      120: SR50_Hori_servo_ctrl.Position:=(OP50_HORI_SERVO_PICK_POS+OP50_Hori_Ser_Jerk_Pos);
	  	   SR50_HORI_servo_ctrl.ABSmove_Start := TRUE;
		   OP50_AutoSeq:=130;

    		   
      130:  SR50_HORI_servo_ctrl.ABSmove_Start := 0;
			SR50_VERT_servo_ctrl.ABSmove_Start := TRUE;	   //MOVING VERTICL SERVO TO SAFE-WORK
            IF OP50_VERT_SERVO_ON_SFE_WRK  THEN
    	      SR50_VERT_servo_ctrl.ABSmove_Start := FALSE;
			  OP50_pick_done:=TRUE;
              OP50_AutoSeq:=140;   
    		END_IF
    		   
      140:  IF (NOT OP50_Gripper_LH_State AND OP50_Grip_LH_Bypass ) AND OP50_Gripper_RH_State THEN  
    			OP50_AutoSeq:=150;
			ELSIF (NOT OP50_Gripper_RH_State AND OP50_Grip_RH_Bypass) AND OP50_Gripper_LH_State THEN
				OP50_AutoSeq:=150;
			ELSIF OP50_Gripper_LH_State AND OP50_Gripper_RH_State THEN  
    			OP50_AutoSeq:=150;
			ELSIF (NOT OP50_Gripper_LH_State AND NOT OP50_Grip_LH_Bypass) OR (NOT OP50_Gripper_RH_State AND NOT OP50_Grip_RH_Bypass) THEN	
				OP50_AutoSeq:=220;
			ELSIF OP50_Grip_LH_Bypass AND OP50_Grip_RH_Bypass THEN
				OP50_AutoSeq:=250;
			END_IF	 
    	    		  
       150:  IF OP50_VERT_SERVO_ON_SFE_WRK  THEN // FEEDING PLACE POSITION TO HORIZONTAL SERVO
    		  SR50_Hori_servo_ctrl.Position:=OP50_HORI_SERVO_PLACE_POS;
              OP50_AutoSeq:=160;				 
    		 END_IF
    		   
       160:  SR50_HORI_servo_ctrl.ABSmove_Start := TRUE;    // MOVING HORIZONTAL SERVO TO PLACE POSITION
    		   IF OP50_HORI_SERVO_ON_WRK_PLACE THEN
    			 SR50_HORI_servo_ctrl.ABSmove_Start := FALSE;
    			 OP50_AutoSeq:=170;
    		   END_IF
       
       170: PAP_CYC_VAR:=0;
			IF OP50_HORI_SERVO_ON_WRK_PLACE AND NOT SR50_VERT_servo_ctrl.ABSmove_Start AND OP50_VERT_SERVO_ON_SFE_WRK AND OP50_STN_ENABLE THEN
    	   	  SR50_Vert_servo_ctrl.Position:=OP50_VERT_SERVO_PLACE_POS;
              OP50_AutoSeq:=175;		
      		END_IF
			
	   175: IF FIXTURE_LH<>40 AND FIXTURE_RH<>40 THEN
		   		OP50_AutoSeq:=250;	
			ELSIF FIXTURE_LH<>40 OR FIXTURE_RH<>40 THEN
				OP50_AutoSeq:=260;	
			ELSE
				OP50_AutoSeq:=180;		
	  	    END_IF
    		
       180: SR50_VERT_servo_ctrl.ABSmove_Start := TRUE; //MOVING VERTICAL SERVO TO PLACE POSITION
    		IF OP50_VERT_SERVO_ON_WRK_PLACE THEN
    			SR50_VERT_servo_ctrl.ABSmove_Start := FALSE;			
				OP50_AutoSeq:=190;				
    		END_IF	
			
       190: IF FIXTURE_LH=40 AND NOT OP50_Grip_LH_Bypass THEN 
				OP50_Gripper_LH_Close:=TRUE;	
			END_IF	
			IF FIXTURE_RH=40 AND NOT OP50_Grip_RH_Bypass THEN 
				OP50_Gripper_RH_Close:=TRUE;	
			END_IF		
			IF Gripper_Aft_Place_Delay.Q THEN	
				OP50_AutoSeq:=200;
			END_IF
			OP50_CURR_MOVER 			:= OP50_STN_MOVER;
			
       200:  //MOVING BACK TO VERTICAL SERVO SAFE POSITION
    		 IF OP50_VERT_SERVO_ON_WRK_PLACE AND NOT SR50_VERT_servo_ctrl.ABSmove_Start THEN
    		   SR50_Vert_servo_ctrl.Position:=OP50_VERT_SERVO_SFE_WRK_POS;
               OP50_AutoSeq:=201; 			   
    		 END_IF
 
	   201: IF Dry_Run THEN
				OP50_AutoSeq:=210; 
			END_IF
			IF  FIXTURE_LH=40 AND FIXTURE_RH=40 THEN
				MOVER_CMP_STATUS[OP50_CURR_MOVER][1]:=50 ;
				MOVER_CMP_STATUS[OP50_CURR_MOVER][2]:=50 ;
				OP50_AutoSeq:=210;
			ELSIF FIXTURE_LH=40 THEN
				MOVER_CMP_STATUS[OP50_CURR_MOVER][1]:=50 ;
				OP50_AutoSeq:=210;
			ELSIF FIXTURE_RH=40 THEN
				MOVER_CMP_STATUS[OP50_CURR_MOVER][2]:=50 ;
				OP50_AutoSeq:=210;
			END_IF		    		 
       210:	  //PROCEEDING FOR NEXT CYCLE
			   SR50_VERT_servo_ctrl.ABSmove_Start := TRUE;           
              IF OP50_VERT_SERVO_ON_SFE_WRK OR OP50_VERT_SERVO_ON_HOME THEN
    			  SR50_VERT_servo_ctrl.ABSmove_Start := FALSE;
				  OP50_STN_ENABLE:=0;				  	  
    			  IF OP50_Gripper_LH_State OR OP50_Gripper_RH_State THEN
    		  		OP50_AutoSeq:=220;
    			  ELSIF (MOVER_CMP_STATUS[OP50_STN_MOVER][1]=50 OR MOVER_CMP_STATUS[OP50_STN_MOVER][2]=50) OR Dry_Run THEN
					STATION_DONE[OP50_CURR_MOVER][OP50_XTS_POS_NO]			:= TRUE;
					IF MOVER_STP_NO[OP50_CURR_MOVER]<>((OP50_XTS_POS_NO*10)+1)THEN
						OP50_AutoSeq:=66;
					END_IF  
				  END_IF				  
    		  END_IF
    		  
       220:  IF (OP50_VERT_SERVO_ON_SFE_WRK OR OP50_VERT_SERVO_ON_HOME OR OP50_VERT_SERVO_ON_WRK_PICK OR OP50_VERT_SERVO_ON_WRK_PLACE) AND NOT SR50_HORI_servo_ctrl.ABSmove_Start AND (OP50_HORI_SERVO_ON_WRK_PLACE OR OP50_HORI_SERVO_ON_WRK_Pick OR OP50_HORI_SERVO_ON_HOME) THEN
    		  SR50_Hori_servo_ctrl.Position:=OP50_HORI_SERVO_SFE_WRK_POS;
			  SR50_Vert_servo_ctrl.Position:=OP50_VERT_SERVO_SFE_WRK_POS;	
              OP50_AutoSeq:=240;			  
    		 END_IF  
    	
       240: SR50_VERT_servo_ctrl.ABSmove_Start := TRUE;
	        IF OP50_VERT_SERVO_ON_SFE_WRK THEN
				SR50_HORI_servo_ctrl.ABSmove_Start := TRUE;
				OP50_AutoSeq:=242;
			 END_IF
			 
	  242: IF OP50_HORI_SERVO_ON_SFE_WRK THEN
    	  	 SR50_HORI_servo_ctrl.ABSmove_Start := FALSE;
      		 OP50_Gripper_RH_Close:=TRUE;	
    		 OP50_Gripper_LH_Close:=TRUE; 	
			 OP50_AutoSeq:=245;		   
      	   END_IF
	 
      245: IF OP50_HORI_SERVO_ON_SFE_WRK AND (NOT OP50_Gripper_LH_State AND NOT OP50_Gripper_RH_State) THEN
    		    OP50_Size_Rej_Complete:=1;
				OP50_AutoSeq:=66;
    	   END_IF
			 
	  250://MOVER_CMP_STATUS[OP50_CURR_MOVER][1]:=51;
		  //MOVER_CMP_STATUS[OP50_CURR_MOVER][2]:=51;
		  OP50_STN_ENABLE:=0;
		  IF (MOVER_CMP_STATUS[OP50_STN_MOVER][1]=51 AND MOVER_CMP_STATUS[OP50_STN_MOVER][2]=51) THEN
			MOVER_STP_NO[OP50_CURR_MOVER]	:= (OP160_XTS_POS_NO*10);
		  ELSE
			STATION_DONE[OP50_CURR_MOVER][OP50_XTS_POS_NO]			:= TRUE;
		  END_IF
		  IF MOVER_STP_NO[OP50_CURR_MOVER]<>((OP50_XTS_POS_NO*10)+1)THEN
			OP50_CURR_MOVER		:= 0;
		  OP50_AutoSeq:=170;	
 		END_IF
		
		
	   260: SR50_Hori_servo_ctrl.Position:=OP50_HORI_SERVO_SFE_WRK_POS;
			SR50_Hori_servo_ctrl.ABSmove_Start:=TRUE;
			IF OP50_HORI_SERVO_ON_SFE_WRK THEN
				OP50_AutoSeq:=270; 
			END_IF
			
	   270: IF FIXTURE_LH<>40 AND NOT OP50_Grip_LH_Bypass THEN
				OP50_Gripper_LH_Close:=TRUE;
				IF NOT OP50_Gripper_LH_State THEN
					OP50_AutoSeq:=280; 
				END_IF
			ELSE
				OP50_AutoSeq:=280;	
			END_IF	
			
	   280: IF FIXTURE_RH<>40 AND NOT OP50_Grip_RH_Bypass THEN
				OP50_Gripper_RH_Close:=TRUE;
				IF NOT OP50_Gripper_RH_State THEN
					OP50_AutoSeq:=290; 
				END_IF
			ELSE
				OP50_AutoSeq:=290;	
			END_IF	

	   290: SR50_Hori_servo_ctrl.Position:=OP50_HORI_SERVO_PLACE_POS;
			SR50_Hori_servo_ctrl.ABSmove_Start:=TRUE;
			IF OP50_HORI_SERVO_ON_WRK_PLACE THEN
				OP50_AutoSeq:=180;	
			END_IF
		
	 300: IF (OP50_HORI_SERVO_ON_SFE_WRK OR OP50_HORI_SERVO_ON_HOME OR OP50_HORI_SERVO_ON_SFE_WRK_PICK ) AND NOT SR50_HORI_servo_ctrl.ABSmove_Start AND OP50_Size_Rej THEN
		  		SR50_Hori_servo_ctrl.Position:=OP50_HORI_SERVO_PICK_POS;
				OP50_Size_Rej_Complete :=0;	
				OP50_Size_Rej          :=0;		
				OP50_AutoSeq:=310;
	       END_IF
		   
	  310: SR50_Hori_servo_ctrl.ABSmove_Start  := TRUE;
		   IF OP50_HORI_SERVO_ON_WRK_PICK THEN
		  		SR50_Vert_servo_ctrl.Position:=OP50_VERT_SERVO_PICK_POS;
				OP50_AutoSeq:=320;
	  	   END_IF
		   
	 320: SR50_VERT_servo_ctrl.ABSmove_Start := TRUE;
		  IF OP50_VERT_SERVO_ON_WRK_PICK THEN
		 	  OP50_Gripper_LH_Open:=OP50_LH_Size_NOK;
			  OP50_Gripper_RH_Open:=OP50_RH_Size_NOK;
			  IF Rejection_Grip_Delay.Q THEN
			  	OP50_AutoSeq:=220;
			  END_IF	
	 	  END_IF	
			
END_CASE

IF OP50_Size_Rej AND OP50_AutoRunning THEN
	OP50_AutoSeq:=300;
END_IF

OP50_STN_ENABLE:=OP50_Continous_Run;

Dry_Run:=All_Station_Dry_Run;
IF Dry_run THEN
	FIXTURE_LH :=40;	
    FIXTURE_RH :=40;
ELSE 
	FIXTURE_LH:=MOVER_CMP_STATUS[OP50_STN_MOVER][1];
	FIXTURE_RH:=MOVER_CMP_STATUS[OP50_STN_MOVER][2];
END_IF

Gripper_Delay(IN:=((OP50_Gripper_RH_State OR OP50_Grip_RH_Bypass) AND (OP50_Gripper_LH_State  OR OP50_Grip_LH_Bypass)),PT:=T#500MS);			
Gripper_pick_Delay(IN:=(OP50_AutoSeq=110),PT:=T#500MS);		
Gripper_Aft_pick_Delay (IN:=(OP50_AutoSeq=110),PT:=T#500MS); 
Gripper_Place_Delay	(IN:=(OP50_AutoSeq=110),PT:=T#500MS);	
Gripper_Aft_Place_Delay(IN:=(OP50_AutoSeq=190),PT:=T#700MS);
	
Rejection_Grip_Delay(IN:=OP50_Size_Rej_Complete,PT:=T#500MS);

del(IN:=tmp,PT:=T#700MS);
IF del.Q THEN
	tmp:=FALSE;
END_IF

//****************Cycle time block*********************************8

OP50_Cycle_Time_FB(i_b_startTime:=OP50_STN_ENABLE , i_b_stopTime:= NOT OP50_STN_ENABLE , o_t_StationTime=>OP50_Cycle_time );					
OP50_PAP_Cycle_Time_FB(i_b_startTime:=PAP_CYC_VAR , i_b_stopTime:= NOT PAP_CYC_VAR , o_t_StationTime=>OP50_PAP_Cycle_time );					
OP50_Overall_Cyc_Time:=OP50_Cycle_time+OP50_PAP_Cycle_time;


////################################ STATION ENABLE CONTION    ############################
OP50_STN_MOVER					:= MOVER_POSITION[OP50_XTS_POS_NO];
	
IF AUTO_WITH_XTS THEN
IF OP50_STN_MOVER>0 THEN
IF NOT(END_OF_CYCLE AND MOVER_CMP_STATUS[OP50_STN_MOVER][1]=5 AND MOVER_CMP_STATUS[OP50_STN_MOVER][2]=5)THEN	
	OP50_STN_ENABLE					:= MOVER_POS_RECHED[OP50_STN_MOVER] AND ((MOVER_CMP_STATUS[OP50_STN_MOVER][1]=40)OR 
										(MOVER_CMP_STATUS[OP50_STN_MOVER][2]=40))AND STATION_ENABLE_CONTROL;	
ELSE
	STATION_DONE[OP50_STN_MOVER][OP50_XTS_POS_NO]			:= TRUE;
END_IF
ELSE
	OP50_STN_ENABLE					:= FALSE;
END_IF	
END_IF

END_PROGRAM

// ---- POUs/Programs/OP50/OP50_Camera_FB.TcPOU
PROGRAM OP50_Camera_FB
VAR
	OP50_LH_Camera 			          : FB_Cognex_ProfiNET_1;

	OP50_LH_Acquisition_Status AT %I*    :Acquisition_Status;
	OP50_LH_Inspection_Status  AT %I*    :Inspection_Status;	
	OP50_LH_Acquisition_ID     AT %I*    :UINT;
	OP50_LH_Inspection_ID   	 AT %I*  :UINT;
	OP50_LH_Error_code      	 AT %I*  :UINT;
	OP50_LH_Current_Job_ID  	 AT %I*  :UINT;
	OP50_LH_Result_code     	 AT %I*  :UINT;
	OP50_LH_Cam_Result      	 AT %I*  :ARRAY[0..63] OF BYTE;	
	OP50_LH_Acquisition_Control AT %Q*  : Acquisition_Control;
	OP50_LH_Inspection_Control  AT %Q*  : Inspection_Control;
	OP50_LH_Command_word		AT %Q*  : UINT;
	OP50_LH_Union                       : UNION_64Byte;
	OP50_LH_Trigger_OK					: BOOL;
	
	OP50_RH_Camera 			          : FB_Cognex_ProfiNET_1;
	
	OP50_RH_Acquisition_Status AT %I*    :Acquisition_Status;
	OP50_RH_Inspection_Status  AT %I*    :Inspection_Status;	
	OP50_RH_Acquisition_ID     AT %I*    :UINT;
	OP50_RH_Inspection_ID   	 AT %I*  :UINT;
	OP50_RH_Error_code      	 AT %I*  :UINT;
	OP50_RH_Current_Job_ID  	 AT %I*  :UINT;
	OP50_RH_Result_code     	 AT %I*  :UINT;
	OP50_RH_Cam_Result      	 AT %I*  :ARRAY[0..63] OF BYTE;	
	OP50_RH_Acquisition_Control AT %Q*  : Acquisition_Control;
	OP50_RH_Inspection_Control  AT %Q*  : Inspection_Control;
	OP50_RH_Command_word		AT %Q*  : UINT;
	OP50_RH_Union                       : UNION_64Byte;
	OP50_RH_Trigger_OK					: BOOL;
END_VAR

OP50_LH_Camera (
	tTimeout:= , 
	sJob_Name:= , 
	camera_ready=> OP50_LH_Camera_Ready,
	Camera_online=> OP50_LH_Camera_Online,
	stCognex_record_status:=OP50_LH_Acquisition_Status, 
	Acquisition_ID:=OP50_LH_Acquisition_ID , 
	stCognex_Inspection_status:=OP50_LH_Inspection_Status, 
	Error_Code:=OP50_LH_Error_code , 
	wcommand_control_in:= OP50_LH_Current_Job_ID, 
	aResults_64_Bytes:= OP50_LH_Cam_Result, 
	number_of_inspections:=OP50_LH_Inspection_ID , 
	iresult_code:= OP50_LH_Result_code, 
	bTarget_job_ID:=OP50_LH_Target_Job_ID , 
	Error_Status_message=> OP50_LH_Error_status, 
	bError=> OP50_LH_Camera_Error, 
	stCognex_record_control=>OP50_LH_Acquisition_Control , 
	stCognex_inspection_control=>OP50_LH_Inspection_Control , 
	wCommandControl_out=>OP50_LH_Command_word , 
	aUser_data_64_Byte=> OP50_LH_Union.aArrayOfByte, 
	bJob_loading_completed=>OP50_LH_Job_Change_Complete , 
	bJob_load_failed=>OP50_LH_Job_Change_Error , 
	bInspection_Result_IO=>  OP50_LH_Trigger_OK, 
	bInspection_Result_NIO=> , 
	bTXTSM_Error_Job_Change=> OP50_LH_Job_Change_Error, 
	bPictureTakenComplete=> OP50_LH_Picture_Taken, 
	Loaded_Job_ID=>OP50_LH_Loaded_Job_ID	 , 
	bClear_Error:= HMI_Reset, 
	bJob_change_start:= OP50_LH_Camera_Job_Change_start, 
	TXTSM_camera_not_online=>OP50_LH_Camera_Error	 , 
	bTrigger_start:= OP50_LH_Camera_Trigger );
	
OP50_RH_Camera (
	tTimeout:= , 
	sJob_Name:= , 
	camera_ready=> OP50_RH_Camera_Ready,
	Camera_online=> OP50_RH_Camera_Online,
	stCognex_record_status:=OP50_RH_Acquisition_Status, 
	Acquisition_ID:=OP50_RH_Acquisition_ID , 
	stCognex_Inspection_status:=OP50_RH_Inspection_Status, 
	Error_Code:=OP50_RH_Error_code , 
	wcommand_control_in:= OP50_RH_Current_Job_ID, 
	aResults_64_Bytes:= OP50_RH_Cam_Result, 
	number_of_inspections:=OP50_RH_Inspection_ID , 
	iresult_code:= OP50_RH_Result_code, 
	bTarget_job_ID:=OP50_RH_Target_Job_ID , 
	Error_Status_message=> OP50_RH_Error_status, 
	bError=> OP50_RH_Camera_Error, 
	stCognex_record_control=>OP50_RH_Acquisition_Control , 
	stCognex_inspection_control=>OP50_RH_Inspection_Control , 
	wCommandControl_out=>OP50_RH_Command_word , 
	aUser_data_64_Byte=> OP50_RH_Union.aArrayOfByte, 
	bJob_loading_completed=>OP50_RH_Job_Change_Complete , 
	bJob_load_failed=>OP50_RH_Job_Change_Error , 
	bInspection_Result_IO=> OP50_RH_Trigger_OK , 
	bInspection_Result_NIO=> , 
	bTXTSM_Error_Job_Change=> OP50_RH_Job_Change_Error, 
	bPictureTakenComplete=> OP50_RH_Picture_Taken, 
	Loaded_Job_ID=>OP50_RH_Loaded_Job_ID	 , 
	bClear_Error:= HMI_Reset, 
	bJob_change_start:= OP50_RH_Camera_Job_Change_start, 
	TXTSM_camera_not_online=>OP50_RH_Camera_Error	 , 
	bTrigger_start:= OP50_RH_Camera_Trigger );

END_PROGRAM

// ---- POUs/Programs/OP50/OP50_Error.TcPOU
PROGRAM OP50_Error
VAR
	OP50_Step_Err_1: TON;
	OP50_Step_Err_2: TON;
	OP50_Step_Err_3: TON;
	OP50_Step_Err_4: TON;
	OP50_Step_Err_5: TON;
	OP50_Step_Err_6: TON;
	
	Gripper_ERR_Timer : TON;
END_VAR

// Set ERROR ACTIVE
IF ((OP50_GVL.OP50_ErrorWord_0<>0) OR (OP50_GVL.OP50_ErrorWord_1<>0) OR (OP50_GVL.OP50_ErrorWord_2<>0)) THEN
	OP50_GVL.OP50_ErrorActive:= TRUE;
END_IF

//Reset ErrorActive
IF OP50_HMI_Reset or HMI_Reset THEN 
	OP50_GVL.OP50_ErrorActive:= FALSE;
	OP50_GVL.OP50_ErrorWord_0:= 0;
	OP50_GVL.OP50_ErrorWord_1:= 0;
	OP50_GVL.OP50_ErrorWord_2:= 0;	
END_IF

// Auto Seq Step Error

//Horizontal Servo is not in home or safe-work position 
OP50_Step_Err_1(IN:=(OP50_GVL.OP50_AutoSeq=70) , PT:=T#5S , Q=> , ET=> );
IF (OP50_GVL.OP50_AutoSeq=70 AND OP50_Step_Err_1.Q) THEN
	OP50_GVL.OP50_ErrorWord_0.0:=TRUE;
END_IF


//Horizontal Servo not reaching pick position 
OP50_Step_Err_1(IN:=(OP50_GVL.OP50_AutoSeq=80) , PT:=T#5S , Q=> , ET=> );
IF (OP50_GVL.OP50_AutoSeq=80 AND NOT OP50_HORI_SERVO_ON_WRK_PICK AND OP50_Step_Err_1.Q) THEN
	OP50_GVL.OP50_ErrorWord_0.1:=TRUE;
END_IF

// Gripper is not closing
OP50_Step_Err_2(IN:=OP50_GVL.OP50_AutoSeq=82 , PT:=T#5S , Q=> , ET=> );
IF (OP50_GVL.OP50_AutoSeq=82 AND OP50_Step_Err_2.Q) THEN
	OP50_GVL.OP50_ErrorWord_0.2:=TRUE;
END_IF

// Vertical Servo not reaching work position 
OP50_Step_Err_3(IN:=OP50_GVL.OP50_AutoSeq=100 , PT:=T#5S , Q=> , ET=> );
IF (OP50_GVL.OP50_AutoSeq=100 AND OP50_Step_Err_3.Q) THEN
	OP50_GVL.OP50_ErrorWord_0.3:=TRUE;
END_IF

// Vertical Servo not reaching safe-work position 
OP50_Step_Err_3(IN:=OP50_GVL.OP50_AutoSeq=150 , PT:=T#5S , Q=> , ET=> );
IF (OP50_GVL.OP50_AutoSeq=150 AND OP50_Step_Err_3.Q) THEN
	OP50_GVL.OP50_ErrorWord_0.4:=TRUE;
END_IF

// Checking the gripper condition is opened or not
OP50_Step_Err_3(IN:=OP50_GVL.OP50_AutoSeq=140 , PT:=T#5S , Q=> , ET=> );
IF (OP50_GVL.OP50_AutoSeq=140 AND OP50_Step_Err_3.Q) THEN
	OP50_GVL.OP50_ErrorWord_0.5:=TRUE;
END_IF

//  Horizontal sevo not moving to place position
OP50_Step_Err_3(IN:=OP50_GVL.OP50_AutoSeq=160 , PT:=T#5S , Q=> , ET=> );
IF (OP50_GVL.OP50_AutoSeq=160 AND OP50_Step_Err_3.Q) THEN
	OP50_GVL.OP50_ErrorWord_0.6:=TRUE;
END_IF

//  Vertical sevo not moving to place position
OP50_Step_Err_3(IN:=OP50_GVL.OP50_AutoSeq=180 , PT:=T#5S , Q=> , ET=> );
IF (OP50_GVL.OP50_AutoSeq=180 AND OP50_Step_Err_3.Q) THEN
	OP50_GVL.OP50_ErrorWord_0.7:=TRUE;
END_IF

// Vertical Servo not reaching safe-work position 
OP50_Step_Err_3(IN:=OP50_GVL.OP50_AutoSeq=210 , PT:=T#5S , Q=> , ET=> );
IF (OP50_GVL.OP50_AutoSeq=210 AND OP50_Step_Err_3.Q) THEN
	OP50_GVL.OP50_ErrorWord_0.8:=TRUE;
END_IF

//  Horizontal sevo not moving to safe work position
OP50_Step_Err_3(IN:=OP50_GVL.OP50_AutoSeq=240 , PT:=T#5S , Q=> , ET=> );
IF (OP50_GVL.OP50_AutoSeq=240 AND OP50_Step_Err_3.Q) THEN
	OP50_GVL.OP50_ErrorWord_0.9:=TRUE;
END_IF

IF Gripper_ERR_Timer.Q THEN
	OP50_GVL.OP50_ErrorWord_0.10:=TRUE;
END_IF

Gripper_ERR_Timer(IN:=I50_LH_GRIP_CLSE_I1101_7 OR I50_RH_GRIP_CLSE_I1110_1,PT:=T#500MS);

END_PROGRAM

// ---- POUs/Programs/OP50/OP50_Initialize_Seq.TcPOU
PROGRAM OP50_Initialize_Seq
VAR
END_VAR

IF OP50_GIUDE_GRP_ctrl.Axis_In_Home AND OP50_GIUDE_GRP_ctrl.Axis_Home_Done AND (SR50_Vert_servo_ctrl.Axis_In_Home) AND OP50_HORI_SERVO_ON_HOME AND NOT I50_LH_GRIP_CLSE_I1101_7 AND  NOT I50_RH_GRIP_CLSE_I1110_1 THEN
	OP50_Temp_hmeOK:=TRUE;
	OP50_HomeRunning:=FALSE;
	OP50_Homing_Seq:=0;
ELSE
	OP50_Temp_hmeOK:=FALSE;	
END_IF

CASE OP50_Homing_Seq OF
	0: IF (OP50_AutoSelected AND NOT OP50_HomeRunning AND NOT OP50_ErrorActive AND NOT OP50_AutoRunning AND NOT OP50_StepRunning AND NOT OP50_Temp_hmeOK) THEN
		OP50_HomeRunning:=TRUE;
		OP50_Homing_Seq:=10;	
	   END_IF
	   
	10:IF (OP50_HomeRunning AND (OP50_HMI_Homing OR HMI_Reset ))THEN 
		IF (SR50_Vert_servo_ctrl.Axis_In_Home) THEN 
			SR50_Vert_servo_ctrl.Axis_Home_Cmd:=FALSE;
		    OP50_Homing_Seq:=20;
		ELSE
			SR50_Vert_servo_ctrl.Position:=0;
			SR50_Vert_servo_ctrl.Velocity:=100;
			SR50_Vert_servo_ctrl.ABSmove_Start:=TRUE;
			SR50_Vert_servo_ctrl.Axis_Home_Cmd:=TRUE;		
	    END_IF
	   END_IF	
	   
   20:  IF (OP50_HORI_SERVO_ON_HOME) THEN 
			SR50_Hori_servo_ctrl.Axis_Home_Cmd:=FALSE;
			OP50_Homing_Seq:=40;
		ELSE
			SR50_Hori_servo_ctrl.Position:=OP50_HORI_SERVO_HME_POS;
			SR50_Hori_servo_ctrl.Velocity:=100;
			SR50_Hori_servo_ctrl.ABSmove_Start:=TRUE;
	    END_IF
		
   40:  CR50_LH_Grip_Cyl.HomingCmd1:=1;
   		CR50_RH_Grip_Cyl.HomingCmd1:=1;
		IF CR50_LH_Grip_Cyl.HomingCmd1 AND CR50_RH_Grip_Cyl.HomingCmd1 THEN
   			OP50_Homing_Seq:=50;
		END_IF	
   
   45:	IF NOT I50_LH_GRIP_CLSE_I1101_7 AND OP50_Gripper_LH_Close THEN 
			OP50_Gripper_LH_State := FALSE;
			OP50_Homing_Seq:=50;
			OP50_Gripper_LH_Close := FALSE;
	    END_IF
				
   50: 	 OP50_Gripper_LH_State := FALSE;
   		 OP50_Gripper_RH_State := FALSE;
   		 OP50_Homing_Seq:=60;
	
   55: 	IF NOT I50_RH_GRIP_CLSE_I1110_1 AND OP50_Gripper_RH_Close THEN 
			OP50_Gripper_RH_State := FALSE;
			OP50_Homing_Seq:=60;
			OP50_Gripper_RH_Close := FALSE;
	    END_IF
		
   60: 	CR50_LH_Rej_Cyl.HomingCmd1:=TRUE;	
		IF CR50_LH_Rej_Cyl.Position1 THEN
			CR50_LH_Rej_Cyl.HomingCmd1:=FALSE;
			OP50_Homing_Seq:=70;
		END_IF
		
   70:	CR50_RH_Rej_Cyl.HomingCmd1:=TRUE;	
		IF CR50_RH_Rej_Cyl.Position1 THEN
			CR50_RH_Rej_Cyl.HomingCmd1:=FALSE;
			OP50_Homing_Seq:=75;
		END_IF
	
  75:	IF OP50_GIUDE_GRP_ctrl.Axis_In_Home AND OP50_GIUDE_GRP_ctrl.Axis_Home_Done THEN
	  		OP50_GIUDE_GRP_ctrl.Bsethome:=0;
			OP50_Homing_Seq:=80;
		ELSE
			OP50_GIUDE_GRP_ctrl.Bsethome:=1;
  		END_IF
	
   80:	OP50_Homing_Seq:=0;
		OP50_HomeRunning:=FALSE;
		OP50_HMI_Homing:=FALSE;
END_CASE

IF NOT OP50_HomeRunning THEN
	   	CR50_LH_Grip_Cyl.HomingCmd1:=0;
		CR50_LH_Rej_Cyl.HomingCmd1:=FALSE;
		CR50_RH_Rej_Cyl.HomingCmd1:=FALSE;
   		CR50_RH_Grip_Cyl.HomingCmd1:=0;
END_IF

END_PROGRAM

// ---- POUs/Programs/OP50/OP50_Conveyor_Cam_Seq.TcPOU
PROGRAM OP50_Conveyor_Cam_Seq
VAR
	OP50_Conveyor_FB	: Servo_Conveyor_FB;
	OP50_Camera_Trigger : BOOL;
	Conveyor_Track_Delay: TON;
	Conveyor_Track_OFF_Delay: TON;
	Conveyor_Continuous_Run: BOOL;
	Conveyor_Velocity_mode: BOOL;
	 OP50_Camera_Trigger_Ack : BOOL;
	Conv_Cam_Step: INT;
	OP50_Miss_Trigger	: BOOL;
	Conv_Temp: BOOL;
	Conv_Step_no: INT;
	Temp_Counter_LH: UINT;
	Temp_Counter_RH: UINT;
	Toggle_Pos_LH : R_TRIG;
	Toggle_Neg_LH : F_TRIG;
	Toggle_Pos_RH : R_TRIG;
	Toggle_Neg_RH : F_TRIG;
	LH_Cam_Completed : BOOL;
	RH_Cam_Completed : BOOL;
	Drum_Jam_Timer	 : TON;
	Toggle_Neg: INT;
	OP50_Camera_Bypass : BOOL;
		Control : BOOL;
END_VAR

Toggle_Pos_LH(CLK:=OP50_Camera_FB.OP50_LH_Inspection_Status.Inspection_Completed);
Toggle_Neg_LH(CLK:=OP50_Camera_FB.OP50_LH_Inspection_Status.Inspection_Completed);
Toggle_Pos_RH(CLK:=OP50_Camera_FB.OP50_RH_Inspection_Status.Inspection_Completed);
Toggle_Neg_RH(CLK:=OP50_Camera_FB.OP50_RH_Inspection_Status.Inspection_Completed);

IF Toggle_Pos_LH.Q OR Toggle_Neg_LH.Q THEN
	LH_Cam_Completed:=1;	
END_IF
IF Toggle_Pos_RH.Q OR Toggle_Neg_RH.Q THEN
	RH_Cam_Completed:=1;	
END_IF


IF MANUAL_SELECTED AND OP50_ManualSelected THEN               
	IF I50_DRUM_CONV_REV_I306_3 THEN
		SR50_Conv_servo_status.targetVelocity:=OP50_Conv_Rev_Speed_6_3;
		SR50_Conv_servo_status.moveVelocity:=I50_DRUM_CONV_REV_I306_3;
 	ELSIF I50_DRUM_CONV_FWD_I306_4 THEN
		SR50_Conv_servo_status.targetVelocity:=OP50_Conv_Fwd_Speed_7_89;
		SR50_Conv_servo_status.moveVelocity:=I50_DRUM_CONV_FWD_I306_4;	
	ELSE 	
		SR50_Conv_servo_status.moveVelocity:=0;   	
	END_IF  	
END_IF

IF OP50_Model='6.3' THEN
	OP50_Conv_Fwd_Time:=OP50_Conv_Fwd_Time_6_3;
	OP50_Conv_Rev_Time:=OP50_Conv_Rev_Time_6_3;
	OP50_Conveyor_FWD_Speed:= OP50_Conv_Fwd_Speed_6_3;
	OP50_Conveyor_REV_Speed:= OP50_Conv_Rev_Speed_6_3;
END_IF

IF OP50_Model='7.89' THEN
	OP50_Conv_Fwd_Time:=OP50_Conv_Fwd_Time_7_89;
	OP50_Conv_Rev_Time:=OP50_Conv_Rev_Time_7_89;
	OP50_Conveyor_FWD_Speed:= OP50_Conv_Fwd_Speed_7_89;
	OP50_Conveyor_REV_Speed:= OP50_Conv_Rev_Speed_7_89;
END_IF

Conveyor_Velocity_mode:=1;

OP50_Conveyor_FB(
	Conveyor_Prgrm_Start:= OP50_AutoRunning, 
	Conveyor_Prgrm_Reset:= , 
	Conveyor_Continuous_Run:= Conveyor_Continuous_Run, 
	Camera_Trigger_OK := OP50_Camera_Done OR OP50_Camera_Bypass, 
	Fwd_Time_IP:= OP50_Conv_Fwd_Time, 
	Rev_Time_IP:= OP50_Conv_Rev_Time, 
	Track_Overflow := Conveyor_Track_OFF_Delay.Q, 
	Track_Sensor_FB := Conveyor_Track_Delay.Q,
	Conveyor_FWD_Position	:= OP50_Conv_Fwd_Pos,
    Conveyor_REV_Position	:= OP50_Conv_Rev_Pos,
    Velocity_mode			:= Conveyor_Velocity_mode,	
	Conveyor_FWD_Speed:=OP50_Conveyor_FWD_Speed , 
	Conveyor_REV_Speed:=OP50_Conveyor_REV_Speed , 
	LH_Work_Sensor:=CR50_LH_Rej_Cyl.Sensor2 , 
	LH_Home_Sensor:=CR50_LH_Rej_Cyl.Sensor1 , 
	RH_Work_Sensor:=CR50_RH_Rej_Cyl.Sensor2 , 
	RH_Home_Sensor:=CR50_RH_Rej_Cyl.Sensor1 , 
	LH_Camera_OK:=  OP50_LH_Camera_OK OR OP50_Camera_Bypass, 
	LH_Camera_NOK:= OP50_LH_Camera_NOK, 
	RH_Camera_OK:=  OP50_RH_Camera_OK OR OP50_Camera_Bypass, 
	RH_Camera_NOK:= OP50_RH_Camera_NOK,
	Step_Num => Conv_Step_no,
	Camera_Trigger_Ack=> OP50_Camera_Trigger_Ack, 
	Camera_trigger:= OP50_Camera_Trigger,
	Drum_ON=> O50_DRUM_MTR_FWD_Q305_5, 
	LH_Work_Coil=>CR50_LH_Rej_Cyl.AutoCmd2 , 
	LH_Home_Coil=>CR50_LH_Rej_Cyl.AutoCmd1 , 
	RH_Work_Coil=>CR50_RH_Rej_Cyl.AutoCmd2,
	RH_Home_Coil=>CR50_RH_Rej_Cyl.AutoCmd1,
	Ready_to_Pick=> OP50_pick_ready , 
	Pick_Done:=     OP50_pick_done , 
	One_Cycle		:= OP50_One_Cycle,
	Conveyor_Servo_Control_Structure:= SR50_CONV_servo_ctrl );

Conveyor_Track_Delay(IN:= NOT I50_DRUM_FEED_CONV1_OVERFLW_I1101_0 OR NOT I50_DRUM_FEED_CONV2_OVERFLW_I1101_1,PT:=INT_TO_TIME(OP50_Drum_ON_Time));	
Conveyor_Track_OFF_Delay(IN:=I50_DRUM_FEED_CONV1_OVERFLW_I1101_0 AND I50_DRUM_FEED_CONV2_OVERFLW_I1101_1,PT:=INT_TO_TIME(OP50_Drum_OFF_Time));  
	
IF 	OP50_AutoRunning OR Conv_Temp THEN
	IF Conveyor_Track_OFF_Delay.Q THEN
		O50_DRUM_MTR_FWD_Q305_5:=0;
	END_IF
	//IF Conveyor_Track_Delay.Q THEN
	//	O50_DRUM_MTR_FWD_Q305_5:=1;
	//END_IF
	O50_AIR_PURGE_ON_Q1153_4:=1;
	O50_DRUM_RUN_IND_Q306_2:=O50_DRUM_MTR_FWD_Q305_5;
ELSE
	O50_DRUM_RUN_IND_Q306_2:=I50_DRUM_OFF_ON_I306_2;
	O50_DRUM_MTR_FWD_Q305_5:=I50_DRUM_OFF_ON_I306_2;
	O50_AIR_PURGE_ON_Q1153_4:=I50_DRUM_OFF_ON_I306_2;
END_IF

IF (NOT OP50_AutoRunning OR (NOT OP50_LH_Camera_Online OR NOT OP50_RH_Camera_Online)) AND NOT OP50_Camera_Bypass THEN
	Conv_Cam_Step:=10;
END_IF 

CASE Conv_Cam_Step OF
	10: 	OP50_LH_Camera_OK :=0;
            OP50_LH_Camera_NOK:=0;
	        OP50_RH_Camera_OK :=0;
	        OP50_RH_Camera_NOK:=0;
			LH_Cam_Completed  :=0;
			RH_Cam_Completed  :=0;			
			OP50_Camera_Done	:=0;
			OP50_LH_Clr_OK 		:=0;
		    OP50_RH_Clr_OK 		:=0;		
			OP50_LH_Size_OK		:=0;
		    OP50_RH_Size_OK		:=0;	
			Conv_Cam_Step		:=11;	
	
	11: IF ((OP50_Camera_Trigger AND (NOT OP50_Camera_Done)) OR OP50_Miss_Trigger) AND NOT OP50_Camera_Bypass THEN
			OP50_LH_Camera_Trigger:=1;
			OP50_RH_Camera_Trigger:=1;
			Conv_Cam_Step		  :=15;	
		END_IF

	15:	IF LH_Cam_Completed AND RH_Cam_Completed THEN// (NOT OP50_LH_Camera_Trigger) AND (NOT OP50_RH_Camera_Trigger) THEN //(Temp_Counter_LH<OP50_Camera_FB.OP50_LH_Acquisition_ID AND Temp_Counter_RH<OP50_Camera_FB.OP50_RH_Acquisition_ID )THEN
			OP50_LH_Camera_Trigger:=0;
			OP50_RH_Camera_Trigger:=0;
			OP50_Camera_Trigger :=0;
			OP50_Miss_Trigger	:=0;
			Conv_Cam_Step:=25;
		END_IF  
	   
	25: IF OP50_Camera_FB.OP50_LH_Cam_Result[0]=1 AND OP50_Camera_FB.OP50_RH_Cam_Result[0]=1 THEN
			OP50_LH_Camera_OK:=1;
			OP50_RH_Camera_OK:=1;
			Conv_Cam_Step    :=50;
		ELSIF (OP50_Camera_FB.OP50_LH_Cam_Result[2]<>1 OR OP50_Camera_FB.OP50_RH_Cam_Result[2]<>1) THEN	
			OP50_One_Cycle  :=1;
			Conv_Cam_Step   :=50;
		ELSIF (OP50_Camera_FB.OP50_LH_Cam_Result[1]=1 OR OP50_Camera_FB.OP50_RH_Cam_Result[1]=1) AND (OP50_Camera_FB.OP50_LH_Cam_Result[2]=1 AND OP50_Camera_FB.OP50_RH_Cam_Result[2]=1) THEN					
			IF OP50_Camera_FB.OP50_LH_Cam_Result[0]=1 THEN
				OP50_LH_Camera_OK:=1;
			END_IF
			IF OP50_Camera_FB.OP50_RH_Cam_Result[0]=1 THEN
				OP50_RH_Camera_OK:=1;
			END_IF
			Conv_Cam_Step:=30;
		END_IF	
			
   30: 	IF OP50_Camera_FB.OP50_LH_Cam_Result[1]=1 THEN
	   		OP50_LH_Camera_NOK:=1;
  	    END_IF
		IF OP50_Camera_FB.OP50_RH_Cam_Result[1]=1 THEN
	   		OP50_RH_Camera_NOK:=1;
  	    END_IF
		Conv_Cam_Step:=50;
		
   50:  OP50_Camera_Done:=1;
   		Temp_Counter_LH:=OP50_Camera_FB.OP50_LH_Acquisition_ID;
		Temp_Counter_RH:=OP50_Camera_FB.OP50_RH_Acquisition_ID;
		IF Conv_Step_no>75 THEN
			Conv_Cam_Step   :=10;
			OP50_Camera_Done:=0;
		END_IF   
END_CASE


IF OP50_AutoRunning AND Control THEN
	Drum_Jam_Timer(IN:=(NOT I50_DRUM_FEED_CONV1_OVERFLW_I1101_0)OR(NOT I50_DRUM_FEED_CONV2_OVERFLW_I1101_1)); 
	Drum_Jam_Timer(PT:=T#40S);
	IF Drum_Jam_Timer.Q THEN
		OP50_ErrorActive:=1;
	END_IF
END_IF

END_PROGRAM

// ---- POUs/Programs/OP60/OP60_MAIN.TcPOU
PROGRAM OP60_MAIN
VAR
	OP60_Modeselection_FB: Mode_Selection_Block1;	
//	OP60_Cycle_Time: Cycle_Time_FB;
	//TP_100ms: TP;
	reset: BOOL;
	Gen_Timer: TON;
END_VAR

// Function Calling

OP60_Manual();
OP60_AUTOSEQUENCE();
OP60_Error();
OP60_Initialization_Seq();
op60_toolchangeover ();
//MOdeselection From HMI

IF (OP60_HMI_AutoMode AND NOT OP60_HMI_ManualMOde AND NOT OP60_HMI_StepMode) THEN
		OP60_Modeselection_FB.ModeWord:=1;
	ELSIF (NOT OP60_HMI_AutoMode AND OP60_HMI_ManualMOde AND NOT OP60_HMI_StepMode) THEN
		OP60_Modeselection_FB.ModeWord:=2;
	ELSIF  (NOT OP60_HMI_AutoMode AND NOT OP60_HMI_ManualMOde AND  OP60_HMI_StepMode) THEN
		OP60_Modeselection_FB.ModeWord:=3;
    ELSE   
		OP60_Modeselection_FB.ModeWord:=0;
END_IF

OP60_Safety_OK:=OperationEnable;

OP60_Modeselection_FB(
	ModeWord:= , 
	HomeConditionOK:=OP60_HomeConditionOK , 
	OperationEnable:=OP60_AutoSelected, 
	StartPB:=OP60_HMI_CycleStart , 
	SafetyAndNOError:= OP60_Safety_OK, 
	ModeAck:=TRUE , 
	HomingINProgress:=OP60_HomeRunning , 
	TempHomeOK:=OP60_Temp_hmeOK , 
	ResetPB:= , 
	AutoSelected=> OP60_AutoSelected, 
	ManualSelected=> OP60_ManualSelected, 
	StepSelected=>OP60_StepSelected , 
	ModeSelAck_Indication=> , 
	StatusDisplay=> , 
	AutoRunning:=OP60_AutoRunning, 
	StepRunning:=OP60_StepRunning , 
	StartEnable:=OP60_StartEnable  , 
	MachineStop:=OP60_Machine_Stop );

OP60_Safety_OK:=OperationEnable;	
	
IF OP60_AutoSelected OR OP60_ManualSelected AND NOT ( OP60_ErrorActive OR OP60_Safety_OK) THEN
	SR60_Vert_servo.bEnable:=TRUE;
ELSE
	SR60_Vert_servo.bEnable:=FALSE;
END_IF

IF OP60_GVL.SR60_Vert_servo.bAxisError OR NOT OP60_Safety_OK  THEN
	OP60_ErrorActive:=TRUE;
END_IF

IF OP60_Stop_Request AND NOT OP60_STN_ENABLE THEN
	OP60_Machine_Stop:=1;
END_IF
Gen_Timer(IN:=OP60_Machine_Stop,PT:=T#5S);
IF Gen_Timer.Q THEN
	OP60_Machine_Stop:=0;
END_IF

END_PROGRAM

// ---- POUs/Programs/OP60/OP60_MANUAL.TcPOU
PROGRAM OP60_MANUAL
VAR
	
    temp_safe:BOOL;
	enable:BOOL;
	reset:bool;
END_VAR


// IF MANUAL IS SELECTED 

//SR60_Vert_servo_ctrl.ABSmove_Start:=OP60_VERT_SERVO_STRT;
OP60_SERVO_POS_DONE:= SR60_Vert_servo_ctrl.pos_done;

IF In_Range(SR60_Vert_servo_status.actualPosition,OP60_VERT_SERVO_SFE_WRK_POS,3) THEN
	OP60_SERVO_ON_SFE_WRK := TRUE;
ELSE
	OP60_SERVO_ON_SFE_WRK := FALSE;
END_IF

IF In_Range(SR60_Vert_servo_status.actualPosition,OP60_VERT_SERVO_HME_POS,1) THEN
	OP60_SERVO_ON_HOME := TRUE;
ELSE
	OP60_SERVO_ON_HOME := FALSE;
END_IF

IF In_Range(SR60_Vert_servo_status.actualPosition,OP60_VERT_SERVO_WRK_POS_1,2) THEN
	OP60_SERVO_ON_WRK_1 := TRUE;
ELSE
	OP60_SERVO_ON_WRK_1 := FALSE;
END_IF

IF In_Range(SR60_Vert_servo_status.actualPosition,OP60_VERT_SERVO_WRK_POS_2,2) THEN
	OP60_SERVO_ON_WRK_2 := TRUE;
ELSE
	OP60_SERVO_ON_WRK_2 := FALSE;
END_IF

OP60_VERT_SERVO_SFE_WRK_POS   :=  OP60_HMI_Safe_Work;
OP60_VERT_SERVO_HME_POS       :=  OP60_HMI_Safe_Home;
OP60_VERT_SERVO_WRK_POS_2     :=  OP60_VERT_SERVO_WORK_POS;
OP60_VERT_SERVO_WRK_POS_1	  := (OP60_VERT_SERVO_WRK_POS_2-OP60_HMI_Servo_Pos_Offset);

SR60_Vert_servo(
	bAxis1_Ref_Switch:= , 
	bInit:= , 
	bErrorReset:= OP60_GVL.OP60_HMI_Reset OR Servo_Reset , 
	bEnable:=Servo_Enable, 
	bMoveVelocity:= , 
	bHalt:= , 
	bManualMode:= MANUAL_SELECTED AND OP60_ManualSelected, 
	fHomePos:= , 
	fOverride:= , 
	fTargetPosition:= SR60_Vert_servo_ctrl.Position, 
	fTargetVelocity:= SR60_Vert_servo_ctrl.Velocity, 
	fAcc:= , 
	fDec:= , 
	Servo_High_Limit:= OP60_HMI_High_Limit,	
	Servo_Low_Limit:=  OP60_HMI_Low_Limit,	
	Safe_move_Conditions:=Servo_Safety,
	Axis:=SR60_Vert_servo_Axis  , 
	bmove_home:=SR60_Vert_servo_ctrl.Axis_Home_Cmd ,
	baxis_in_home_pos=>SR60_Vert_servo_ctrl.Axis_In_Home ,
	HME_WRITE_ADD:= 16#5018, 
	bHome:=SR60_Vert_servo_ctrl.Bsethome , 
	bSetPosition:=SR60_Vert_servo_ctrl.BsetPos , 
	bMoveAbsolute:=SR60_Vert_servo_ctrl.ABSmove_Start , 
	bMoveTorque :=SR60_Vert_servo_ctrl.Torque_mode_Start,	
	bMoveRelative:=SR60_Vert_servo_ctrl.RELmove_Start , 
	stManualModeAxis:=SR60_Vert_servo_status , 
	sAxisState=>SR60_Vert_servo_ctrl.Axis_State , 
	bAxis_ready=>SR60_Vert_servo_ctrl.Axis_ready , 
	bAxisInPosition=> SR60_Vert_servo_ctrl.Axis_In_Pos, 
	bAxisError=>SR60_Vert_servo_ctrl.Axis_Error , 
	bAxisEnabled=> SR60_Vert_servo_ctrl.Axis_Enabled, 
	bAxisHomed=> SR60_Vert_servo_ctrl.Axis_reference, 
	bSetPositionDone=>   ,
    bsafe_to_move=>SR60_Vert_servo_ctrl.Safe_To_Move,  
	bABS_Pos_done=> SR60_Vert_servo_ctrl.pos_done,
	bHaltDone=> , 
	bSTOPDone=> , 
	bHomeDone=> , 
	bDone=> ,
	Actual_position=>SR60_Vert_servo_ctrl.Actual_Position ,  
	Actual_velocity=>SR60_Vert_servo_ctrl.Actual_Velocity , 
	Actual_Torque=> SR60_Vert_servo_ctrl.Actual_Torque);
	
IF MANUAL_SELECTED and OP60_ManualSelected THEN
	SR60_Vert_servo_status.targetVelocity:=250;	
END_IF	
	

OP60_LH_LVDT_VALUE := DINT_TO_REAL(OP60_LH)/10000;
OP60_RH_LVDT_VALUE := DINT_TO_REAL(OP60_RH)/10000;

END_PROGRAM

// ---- POUs/Programs/OP60/OP60_AUTOSEQUENCE.TcPOU
PROGRAM OP60_AUTOSEQUENCE
VAR

//INT

	OP60_FIXTURE_2					: INT;
	OP60_FIXTURE_1					: INT;	
	
// TIMER
	OP60_AFT_WRK_POS : TON;
	dry_run : BOOL;
	check: BOOL;

	OP60_STN_MOVER: INT;
	MOVER_POS_RECHED_R: R_TRIG;
	OP60_Cycle_Time_FB : FB_Cycletime;
END_VAR

VAR PERSISTENT
	
END_VAR

IF (NOT OP60_AutoSelected) OR (OP60_ErrorActive OR OP60_HomeRunning ) OR NOT OperationEnable THEN
	OP60_AutoRunning:= FALSE;
	OP60_AutoSeq:= 10;
	OP60_STN_ENABLE:=FALSE;
END_IF	

CASE OP60_AutoSeq OF
		
		10: IF (OP60_AutoSelected) THEN		// Check Automode Selected
				OP60_AutoSeq:=20;
	        END_IF
		
	    20:IF ( NOT OP60_ErrorActive) THEN		//Check No error
		       OP60_AutoSeq:=30;
      	   END_IF
		   
      	30:IF (NOT OP60_HomeRunning) THEN		//Check No Homerunning
      		   OP60_AutoSeq :=40;
      	   END_IF
		   
        40:IF (OP60_Main.OP60_Modeselection_FB.TempHomeOK)THEN	//Check Machine in Home
      		   OP60_AutoSeq:= 50;
      	   END_IF
		   
      	50:IF ( OP60_STN_ENABLE AND OP60_STN_RUNNING ) THEN		// Check Operation Completed Reset
      		   OP60_AutoSeq:=70;
		   ELSE
	   		   OP60_AutoSeq:=60;
      	   END_IF
		   
	   60:IF (AUTO_RUNNING OR (NOT AUTO_RUNNING AND OP60_HMI_CycleStart)) THEN		//Machine Start in Fully Automatic or Press Cycle Start For Semi Automatic
		    OP60_HomeConditionOK:=TRUE;
	 			IF( OP60_Main.OP60_Modeselection_FB.HomeConditionOK AND OP60_AutoSelected) THEN
					OP60_AutoRunning:=TRUE;
					OP60_StepRunning:= FALSE;		
				ELSIF (OP60_Main.OP60_Modeselection_FB.HomeConditionOK AND OP60_StepSelected) THEN
					OP60_AutoRunning:=FALSE;
					OP60_StepRunning:= TRUE;
				END_IF;
		  END_IF
		  
		  IF ((OP60_AutoRunning OR OP60_StepRunning) AND OP60_StartEnable) THEN
			OP60_AutoSeq:= 70;
		  END_IF	

      	70:  // SERVO POSITION SAFE CHECK
	       IF (OP60_SERVO_ON_SFE_WRK OR OP60_SERVO_ON_HOME) AND NOT SR60_Vert_servo_ctrl.ABSmove_Start THEN 
	        SR60_Vert_servo_ctrl.Position:=OP60_VERT_SERVO_WRK_POS_1;   
	        OP60_AutoSeq:=75;
	       END_IF
		   
		75: // WAITING FOR MOVER AND MOVING SERVO TO TARGET POSITION
			IF OP60_STN_ENABLE AND SR60_Vert_servo_ctrl.Position=OP60_VERT_SERVO_WRK_POS_1 THEN
			 SR60_Vert_servo_ctrl.Velocity:=OP60_HMI_Servo_Speed;
			 OP60_STN_RUNNING:=1;
			 SR60_Vert_servo_ctrl.ABSmove_Start:=TRUE;
			 IF OP60_FIXTURE_1=50 OR OP60_FIXTURE_2=50 THEN
			 	OP60_AutoSeq:=60;
			 ELSIF OP60_FIXTURE_1<>50 AND OP60_FIXTURE_2<>50 THEN
				OP60_AutoSeq:=76;
			 END_IF		
			END_IF
			
	 76:	OP60_STN_ENABLE:=0;
			IF 	(MOVER_CMP_STATUS[OP60_STN_MOVER][1]=51 AND MOVER_CMP_STATUS[OP60_STN_MOVER][2]=51) THEN
				MOVER_STP_NO[OP60_CURR_MOVER]	:= (OP160_XTS_POS_NO*10);
			ELSE		
				STATION_DONE[OP60_CURR_MOVER][OP60_XTS_POS_NO]	:= TRUE;
			END_IF	
			IF MOVER_STP_NO[OP60_CURR_MOVER]<>((OP60_XTS_POS_NO*10)+1)THEN 
				OP60_CURR_MOVER	:= 0;
				OP60_AutoSeq	:=75;  
			END_IF	
			
		80:  IF SR60_Vert_servo_ctrl.pos_done AND OP60_SERVO_ON_WRK_1 THEN
			   SR60_Vert_servo_ctrl.ABSmove_Start:=FALSE;
			   SR60_Vert_servo_ctrl.Position:=OP60_GVL.OP60_VERT_SERVO_WRK_POS_2;
			   SR60_Vert_servo_ctrl.Velocity:=(OP60_HMI_Servo_Speed-OP60_HMI_Servo_Speed_Offset);
			   OP60_AutoSeq:=90;
			 ELSIF SR60_Vert_servo_ctrl.pos_done AND OP60_SERVO_ON_WRK_2 THEN
 				OP60_AutoSeq:=100;
			 END_IF
			  
		90: IF OP60_SERVO_ON_WRK_1 AND NOT SR60_Vert_servo_ctrl.ABSmove_Start THEN 
				OP60_LH_LVDT_OK:=0;
				OP60_LH_LVDT_NOK:=0;
				OP60_RH_LVDT_OK:=0;
				OP60_RH_LVDT_NOK:=0;	                  
               SR60_Vert_servo_ctrl.ABSmove_Start:=TRUE; 
               OP60_AutoSeq:=100;
			END_IF
			
		100: // START THE SPINNER OK COMPONENT FIXTURE
			IF OP60_AFT_WRK_POS.Q AND OP60_SERVO_ON_WRK_2 THEN	
			 SR60_Vert_servo_ctrl.ABSmove_Start:=FALSE;		 
			  IF OP60_FIXTURE_1=50 THEN
			 	 IF In_Range(OP60_LH_LVDT_VALUE,OP60_SET_LVDT_VALUE,OP60_LVDT_TOLERANCE) THEN
				  OP60_LH_LVDT_OK  := 1;
				  OP60_LH_LVDT_NOK := 0;				  				  
			 	 ELSE
				  OP60_LH_LVDT_NOK := 1;
				  OP60_LH_LVDT_OK  := 0;
			 	 END_IF  
			  END_IF
			  IF OP60_FIXTURE_2=50 THEN
			  	IF In_Range(OP60_RH_LVDT_VALUE,OP60_SET_LVDT_VALUE,OP60_LVDT_TOLERANCE) THEN
				  OP60_RH_LVDT_OK  := 1;
				  OP60_RH_LVDT_NOK := 0;			  				  
			  	ELSE
				  OP60_RH_LVDT_NOK := 1;
				  OP60_RH_LVDT_OK  := 0;
			    END_IF
		 	  END_IF
				OP60_HMI_LH_LVDT_VALUE:=OP60_LH_LVDT_VALUE;
				OP60_HMI_RH_LVDT_VALUE:=OP60_RH_LVDT_VALUE;	
			  IF NOT SR60_Vert_servo_ctrl.ABSmove_Start THEN
				 SR60_Vert_servo_ctrl.Position:=OP60_VERT_SERVO_SFE_WRK_POS;
				 SR60_Vert_servo_ctrl.Velocity:=OP60_HMI_Servo_Speed;
				 OP60_AutoSeq:=110;
			  END_IF				    			  
		    END_IF
			OP60_CURR_MOVER				:= OP60_STN_MOVER;
		
		110: // SERVO MOVE TO SAFE WORK POSITION	 
			IF NOT SR60_Vert_servo_ctrl.ABSmove_Start AND SR60_Vert_servo.fTargetPosition=OP60_VERT_SERVO_SFE_WRK_POS THEN
				SR60_Vert_servo_ctrl.ABSmove_Start:=TRUE;
				IF OP60_LH_LVDT_OK THEN
					MOVER_CMP_STATUS[OP60_CURR_MOVER][1]:=60;
				ELSIF OP60_LH_LVDT_NOK THEN  
					MOVER_CMP_STATUS[OP60_CURR_MOVER][1]:=61;	
				END_IF
				IF OP60_RH_LVDT_OK THEN
					MOVER_CMP_STATUS[OP60_CURR_MOVER][2]:=60;
				ELSIF OP60_RH_LVDT_NOK THEN  
					MOVER_CMP_STATUS[OP60_CURR_MOVER][2]:=61;	
				END_IF	
				OP60_STN_ENABLE:=FALSE;				
				OP60_AutoSeq:=120;
			END_IF

				
		120: // SERVO DONE
			IF SR60_Vert_servo_ctrl.pos_done AND OP60_SERVO_ON_SFE_WRK THEN
			 	SR60_Vert_servo_ctrl.ABSmove_Start:=FALSE;
			 	OP60_AutoSeq:=70;			
				OP60_STN_RUNNING:=0;
		  IF (MOVER_CMP_STATUS[OP60_STN_MOVER][1]=61 AND MOVER_CMP_STATUS[OP60_STN_MOVER][2]=61) THEN
			MOVER_STP_NO[OP60_CURR_MOVER]	:= (OP160_XTS_POS_NO*10);
			ELSE
				STATION_DONE[OP60_CURR_MOVER][OP60_XTS_POS_NO]			:= TRUE;	
			 	OP60_STN_ENABLE:=FALSE;
			END_IF	
			END_IF		
END_CASE 


OP60_Cycle_Time_FB(i_b_startTime:=OP60_STN_ENABLE , i_b_stopTime:= NOT OP60_STN_ENABLE , o_t_StationTime=>OP60_Cycle_time );					

OP60_AFT_WRK_POS(IN:=(OP60_SERVO_ON_WRK_2 AND (OP60_AutoSeq=100)), PT:=INT_TO_TIME(OP60_DLY_AFT_SFE_WRK) , Q=> , ET=> );
//Timer(IN:=OP60_STN_ENABLE,PT:=T#10S);
Dry_Run:=All_Station_Dry_Run;
IF dry_run THEN
	OP60_FIXTURE_1:=50;	
	OP60_FIXTURE_2:=50;
ELSE
	OP60_FIXTURE_1:=MOVER_CMP_STATUS[OP60_STN_MOVER][1];
	OP60_FIXTURE_2:=MOVER_CMP_STATUS[OP60_STN_MOVER][2];	
END_IF


//#######################      OP60 ENABLE CONDITION	#########################

	OP60_STN_MOVER					:= MOVER_POSITION[OP60_XTS_POS_NO];
IF AUTO_WITH_XTS THEN
IF OP60_STN_MOVER>0 THEN	
IF NOT(END_OF_CYCLE AND MOVER_CMP_STATUS[OP60_STN_MOVER][1]=5 AND MOVER_CMP_STATUS[OP60_STN_MOVER][2]=5)THEN	
	OP60_STN_ENABLE					:= MOVER_POS_RECHED[OP60_STN_MOVER] AND ((MOVER_CMP_STATUS[OP60_STN_MOVER][1]=50)OR 
										(MOVER_CMP_STATUS[OP60_STN_MOVER][2]=50)) AND STATION_ENABLE_CONTROL;
ELSE
	STATION_DONE[OP60_STN_MOVER][OP60_XTS_POS_NO]			:= TRUE;		
END_IF
ELSE
	OP60_STN_ENABLE					:= FALSE;
END_IF	
END_IF

END_PROGRAM

// ---- POUs/Programs/OP60/OP60_ERROR.TcPOU
PROGRAM OP60_ERROR
VAR
	OP60_StepErr_1: TON;
	OP60_Step_Err_2: TON;
END_VAR

// Set ERROR ACTIVE
IF ((OP60_GVL.OP60_ErrorWord_0<>0) OR (OP60_GVL.OP60_ErrorWord_1<>0) OR (OP60_GVL.OP60_ErrorWord_2<>0)) THEN
	OP60_GVL.OP60_ErrorActive:= TRUE;
	END_IF

//Reset ErrorActive
IF (OP60_HMI_Reset OR HMI_Reset) THEN 
	OP60_GVL.OP60_ErrorActive:= FALSE;
	OP60_GVL.OP60_ErrorWord_0:= 0;
	OP60_GVL.OP60_ErrorWord_1:= 0;
	OP60_GVL.OP60_ErrorWord_2:= 0;

END_IF

OP60_ErrorWord_0.0:=SR60_Vert_servo.bAxisError;
OP60_ErrorWord_0.1:=NOT OperationEnable;

// Auto Seq Step Error
//Servo not reaching work position
OP60_StepErr_1(IN:=(OP60_AutoSeq=80) , PT:=T#5S , Q=> , ET=> );
IF (OP60_AutoSeq=80 AND NOT OP60_GVL.OP60_SERVO_ON_WRK_1 AND OP60_StepErr_1.Q) THEN
	OP60_GVL.OP60_ErrorWord_0.2:=TRUE;
END_IF

// Servo Not Reached home position or safe-work position
OP60_Step_Err_2(IN:=OP60_AutoSeq=120 , PT:=T#5S , Q=> , ET=> );
IF (OP60_AutoSeq=120 AND NOT SR60_Vert_servo_ctrl.Axis_In_Home AND OP60_Step_Err_2.Q) THEN
	OP60_GVL.OP60_ErrorWord_0.3:=TRUE;
END_IF

//OP20_StepErr_3(IN:=( OP60_HomeRunning AND (OP60_Homing_Seq=10)), PT:=T#5S , Q=> , ET=> );
//IF OP20_StepErr_3.Q THEN
//	OP20_GVL.OP20_ErrorWord_0.4:=TRUE;
//END_IF

END_PROGRAM

// ---- POUs/Programs/OP60/OP60_Initialization_Seq.TcPOU
PROGRAM OP60_Initialization_Seq
VAR
END_VAR

IF (SR60_Vert_servo_ctrl.Axis_In_Home)THEN
    OP60_Temp_hmeOK:=TRUE;
	OP60_HomeRunning:=FALSE;
	OP60_Homing_Seq:=0;
ELSE
	OP60_Temp_hmeOK:=FALSE;	
END_IF

CASE OP60_Homing_Seq OF
	0: IF (OP60_AutoSelected AND NOT OP60_HomeRunning AND NOT OP60_ErrorActive AND NOT  OP60_AutoRunning AND NOT OP60_StepRunning AND NOT OP60_Temp_hmeOK ) THEN
		OP60_HomeRunning:=TRUE;
		OP60_Homing_Seq:=10;	
	   END_IF
	10:IF (OP60_HomeRunning AND (OP60_HMI_Homing OR HMI_Reset))THEN 
		IF (SR60_Vert_servo_ctrl.Axis_In_Home) THEN 
			OP60_Homing_Seq:=20;
			SR60_Vert_servo_ctrl.Axis_Home_Cmd:=FALSE;
		ELSE
			SR60_Vert_servo_ctrl.Position:=0;
			SR60_Vert_servo_ctrl.Velocity:=100;			
			SR60_Vert_servo_ctrl.ABSmove_Start:=TRUE;
			SR60_Vert_servo_ctrl.Axis_Home_Cmd:=TRUE;
	    END_IF
	   END_IF		
	20:	OP60_Homing_Seq:=0;
		OP60_HomeRunning:=FALSE;
	
END_CASE

END_PROGRAM

// ---- POUs/Programs/OP60/op60_toolchangeover.TcPOU
PROGRAM op60_toolchangeover
VAR
	op60_tool_change                    : tool_changeover;
	OP60_TOOL_CHANGE_MODE_SELECTED      : BOOL;
	fb_reset_1                          : BOOL;
	tool_6_fb                           : BOOL;
	tool_8_fb                           : BOOL;
	OP60_TOL_UNLOD_STRT					: BOOL;
	OP60_TOL_LOAD_STRT					: BOOL;
	OP60_TOL_DISENGAGE					: BOOL;
	OP60_TOL_ENGAGE						: BOOL;
	op60_manual_lock                    : BOOL;
	op60_manual_unlock                  : BOOL;
	OP60_UNLD_STUS                      : STRING;
	OP60_LOAD_STUS                      : STRING;
END_VAR

VAR PERSISTENT
	
	OP60_TOL_WRK_POS					: LREAL;
	OP60_TOL_HME_POS					: LREAL;
	op60_TOL_VELOCITY					: LREAL;
	OP60_TOL_CHNGE_CMPLE				: BOOL;
	OP60_TOL_LOAD_COMPLE                : BOOL;
	OP60_TOL_UNLOAD_COMPLE              : BOOL;
	
END_VAR

IF OP60_TOOL_CHANGE_MODE_SELECTED THEN

op60_tool_change(
	actual_pos:=SR60_Vert_servo_ctrl.Actual_Position,
	actual_vel:=SR60_Vert_servo_ctrl.Actual_Velocity,
	target_work_pos:= OP60_TOL_WRK_POS, 
	target_home_pos:= OP60_TOL_HME_POS, 
	target_vel_from_hmi:= op60_TOL_VELOCITY, 
	station_number:= , 
	mover_number:= , 
	no_of_mover_present:= , 
	model_selected:= model_selected, 
	tool_unloading_start:=OP60_TOL_UNLOD_STRT , 
	tool_loading_start:=OP60_TOL_LOAD_STRT , 
	error_active:= , 
	station_in_auto:= OP60_AutoSelected,                   
	station_in_home:=  ,                                   
	absoulte_move_done:= SR60_Vert_servo_ctrl.Axis_In_Pos, 
	tool_6_3_present:= tool_6_fb, 
	tool_7_89_present:= tool_8_fb, 
	fb_reset:=fb_reset_1,
	SERVO_TOL_CHECK_OFFSET_POS := 18, 
	tool_changer_over_complete=> OP60_TOL_CHNGE_CMPLE,
	tool_disengage=> OP60_TOL_DISENGAGE, 
	tool_engagae=> OP60_TOL_ENGAGE, 
	tool_loading_complete=> OP60_TOL_LOAD_COMPLE, 
	tool_unloading_complete=> OP60_TOL_UNLOAD_COMPLE, 
	servo_move_abs=>SR60_Vert_servo_ctrl.ABSmove_Start, 
	unloading_status=>OP60_UNLD_STUS , 
	loading_status=>OP60_LOAD_STUS , 
	target_pos_to_servo=>SR60_Vert_servo_ctrl.Position, 
	target_vel_to_servo=>SR60_Vert_servo_ctrl.Velocity,
    tool_loading_failed := );
	
END_IF	

IF op60_manual_lock OR OP60_TOL_ENGAGE THEN
	O60_TOOL_CHO_UNLOCK_Q1152_2  :=0;
	O60_TOOL_CHO_LOCK_Q1152_3    :=1;
ELSIF op60_manual_unlock OR OP60_TOL_DISENGAGE THEN
	O60_TOOL_CHO_UNLOCK_Q1152_2  :=0;
	O60_TOOL_CHO_LOCK_Q1152_3    :=1;
END_IF

END_PROGRAM

// ---- POUs/Programs/OP70/OP70_MAIN.TcPOU
PROGRAM OP70_MAIN
VAR
	OP70_Modeselection_FB: Mode_Selection_Block1;
	TP_100ms: TP;
	Pulse_1s: BOOL;
	Times: LREAL;
	Pge_NUM : INT;
	Gen_Timer: TON;
END_VAR


OP70_Manual();
OP70_AUTOSEQUENCE();
//OP70_CONVEYOR();
OP70_Camera_FB();
OP70_Error();
OP70_Initialize_Seq();
OP70_Conveyor_Cam_Seq();
//MOdeselection From HMI

IF (OP70_GVL.OP70_HMI_AutoMode AND NOT OP70_GVL.OP70_HMI_ManualMOde AND NOT OP70_GVL.OP70_HMI_StepMode) THEN
	OP70_Modeselection_FB.ModeWord:=1;
	ELSIF (NOT OP70_GVL.OP70_HMI_AutoMode AND OP70_GVL.OP70_HMI_ManualMOde AND NOT OP70_GVL.OP70_HMI_StepMode) THEN
		OP70_Modeselection_FB.ModeWord:=2;
	ELSIF  (NOT OP70_GVL.OP70_HMI_AutoMode AND NOT OP70_GVL.OP70_HMI_ManualMOde AND  OP70_GVL.OP70_HMI_StepMode) THEN
		OP70_Modeselection_FB.ModeWord:=3;
    ELSE   
		OP70_Modeselection_FB.ModeWord:=0;
END_IF
(*
IF  (OP70_AutoSelected OR OP70_ManualSelected ) AND NOT OP70_ErrorActive AND OP70_Safety_OK THEN
  SR70_CONV_servo.bEnable:=TRUE;
  SR70_HORI_servo.bEnable:=TRUE;
  SR70_VERT_servo.bEnable:=TRUE;
ELSE 
  SR70_CONV_servo.bEnable:=FALSE;
  SR70_HORI_servo.bEnable:=FALSE;
  SR70_VERT_servo.bEnable:=FALSE;	
END_IF*)

IF SR70_CONV_servo.bAxisError OR SR70_HORI_servo.bAxisError OR SR70_VERT_servo.bAxisError THEN
	OP70_ErrorActive:=TRUE;
END_IF

OP70_Safety_OK:=OperationEnable;

OP70_Modeselection_FB(
	ModeWord:= , 
	HomeConditionOK:=OP70_HomeConditionOK , 
	OperationEnable:=OP70_AutoSelected AND OP70_Safety_OK , 
	StartPB:=OP70_HMI_Cycle_Start , 
	SafetyAndNOError:= OP70_Safety_OK, 
	ModeAck:=TRUE , 
	HomingINProgress:=OP70_HomeRunning , 
	TempHomeOK:=OP70_Temp_hmeOK , 
	ResetPB:= , 
	AutoSelected=> OP70_AutoSelected, 
	ManualSelected=> OP70_ManualSelected, 
	StepSelected=>OP70_StepSelected , 
	ModeSelAck_Indication=> , 
	StatusDisplay=> , 
	AutoRunning:=OP70_AutoRunning, 
	StepRunning:=OP70_StepRunning , 
	StartEnable:=OP70_StartEnable  , 
	MachineStop:=OP70_Machine_Stop );

IF OP70_Stop_Request AND NOT OP70_STN_ENABLE THEN
	OP70_Machine_Stop:=1;
END_IF
Gen_Timer(IN:=OP70_Machine_Stop,PT:=T#5S);
IF Gen_Timer.Q THEN
	OP70_Machine_Stop:=0;
END_IF

END_PROGRAM

// ---- POUs/Programs/OP70/OP70_MANUAL.TcPOU
PROGRAM OP70_MANUAL
VAR
	SR70_Vert_servo_Axis :AXIS_REF;
	SR70_Hori_servo_Axis :AXIS_REF;
	SR70_Conv_servo_Axis :AXIS_REF;
	SR70_GUIDE_GRP_AXIS :AXIS_REF;
	LH_Gripper_bMove	 : BOOL;
	RH_Gripper_bMove	 : BOOL;
	
	temp_safe: BOOL;
	temp:BOOL;

	error70: BOOL;
	OP70Enable: BOOL;
	FESTO_NOT_NEED: BOOL;
	NOT_REQ: BOOL;
	OP70EnableHorz: BOOL;
	Grip_Test: INT;
	Test: TON;
	A1: BOOL;
	A2: BOOL;

END_VAR


OP70_VERT_SERVO_POSITION    := SR70_Vert_servo_ctrl.Actual_Position;
OP70_VERT_SERVO_POS_DONE	:= SR70_Vert_servo_ctrl.pos_done ;

OP70_HORI_SERVO_POSITION    := SR70_Hori_servo_ctrl.Actual_Position;
OP70_HORI_SERVO_POS_DONE	:= SR70_Hori_servo_ctrl.pos_done ;

OP70_CONV_SERVO_POSITION    := SR70_CONV_servo_ctrl.Actual_Position;
OP70_CONV_SERVO_POS_DONE	:= SR70_CONV_servo_ctrl.pos_done ;


// VERTICAL SERVO 
IF In_Range(SR70_Vert_servo_status.actualPosition,OP70_VERT_SERVO_SFE_WRK_POS,1) THEN
	OP70_VERT_SERVO_ON_SFE_WRK := TRUE;
ELSE
	OP70_VERT_SERVO_ON_SFE_WRK := FALSE;
END_IF

IF In_Range(SR70_Vert_servo_status.actualPosition,OP70_VERT_SERVO_HME_POS,1) THEN
	OP70_VERT_SERVO_ON_HOME := TRUE;
ELSE
	OP70_VERT_SERVO_ON_HOME := FALSE;
END_IF

IF In_Range(SR70_Vert_servo_status.actualPosition,OP70_VERT_SERVO_PICK_POS,1) THEN
	OP70_VERT_SERVO_ON_WRK_PICK := TRUE;
ELSE
	OP70_VERT_SERVO_ON_WRK_PICK := FALSE;
END_IF		

IF In_Range(SR70_Vert_servo_status.actualPosition,OP70_VERT_SERVO_PLACE_POS,1) THEN
	OP70_VERT_SERVO_ON_WRK_PLACE := TRUE;
ELSE
	OP70_VERT_SERVO_ON_WRK_PLACE := FALSE;
END_IF

//HORIZONTAL SERVO
IF In_Range(SR70_Hori_servo_status.actualPosition,OP70_HORI_SERVO_SFE_WRK_POS,1) THEN
	OP70_HORI_SERVO_ON_SFE_WRK := TRUE;
ELSE
	OP70_HORI_SERVO_ON_SFE_WRK := FALSE;
END_IF

IF In_Range(SR70_Hori_servo_status.actualPosition,OP70_HORI_SERVO_HME_POS,1) THEN
	OP70_HORI_SERVO_ON_HOME := TRUE;
ELSE
	OP70_HORI_SERVO_ON_HOME := FALSE;
END_IF

IF In_Range(SR70_Hori_servo_status.actualPosition,OP70_HORI_SERVO_PICK_POS,4) THEN
	OP70_HORI_SERVO_ON_WRK_PICK := TRUE;
ELSE
	OP70_HORI_SERVO_ON_WRK_PICK := FALSE;
END_IF	

IF In_Range(SR70_Hori_servo_status.actualPosition,OP70_HORI_SERVO_SAFE_PICK_POS,1) THEN
	OP70_HORI_SERVO_ON_SFE_WRK_PICK := TRUE;
ELSE
	OP70_HORI_SERVO_ON_SFE_WRK_PICK := FALSE;
END_IF	

IF In_Range(SR70_Hori_servo_status.actualPosition,OP70_HORI_SERVO_PLACE_POS,1) THEN
	OP70_HORI_SERVO_ON_WRK_PLACE := TRUE;
ELSE
	OP70_HORI_SERVO_ON_WRK_PLACE := FALSE;
END_IF	

//CONVEYOR SERVO

IF In_Range(SR70_CONV_servo_status.actualPosition,OP70_CONV_SERVO_SFE_WRK_POS,1) THEN
	OP70_CONV_SERVO_ON_SFE_WRK := TRUE;
ELSE
	OP70_CONV_SERVO_ON_SFE_WRK := FALSE;
END_IF

IF In_Range(SR70_CONV_servo_status.actualPosition,OP70_CONV_SERVO_HME_POS,1) THEN
	OP70_CONV_SERVO_ON_HOME := TRUE;
ELSE
	OP70_CONV_SERVO_ON_HOME := FALSE;
END_IF

IF In_Range(SR70_CONV_servo_status.actualPosition,OP70_CONV_SERVO_WRK_POS,1) THEN
	OP70_CONV_SERVO_ON_WRK := TRUE;
ELSE
	OP70_CONV_SERVO_ON_WRK := FALSE;
END_IF	


OP70_GVL.SR70_Vert_servo(
	bAxis1_Ref_Switch:= temp, 
	bInit:= , 
	bErrorReset:=OP70_HMI_Reset OR Servo_Reset , 
	bEnable:= Servo_Enable, 
	bMoveVelocity:= , 
	bHalt:= , 
	bManualMode:= OP70_ManualSelected AND MANUAL_SELECTED ,
	fHomePos:= , 
	fOverride:= , 
	fTargetPosition:=SR70_Vert_servo_ctrl.Position , 
	fTargetVelocity:=SR70_Vert_servo_ctrl.Velocity , 
	fAcc:= , 
	fDec:= ,
	Servo_High_Limit:= OP70_HMI_Vert_High_Limit,	
	Servo_Low_Limit:= OP70_HMI_Vert_Low_Limit,	 	
	WARNING_LIMIT:=1,	
	Actual_Torque=> SR70_Vert_servo_ctrl.Actual_Torque ,
	Actual_position=>SR70_Vert_servo_ctrl.Actual_Position ,
    Actual_velocity=>SR70_Vert_servo_ctrl.Actual_Velocity ,	
	bmove_home:=SR70_Vert_servo_ctrl.Axis_Home_Cmd ,
	baxis_in_home_pos=>SR70_Vert_servo_ctrl.Axis_In_Home ,
	Safe_move_Conditions:=Servo_Safety,
	Axis:= SR70_Vert_servo_Axis , 
	HME_WRITE_ADD:= 16#500C,	
	bHome:=SR70_Vert_servo_ctrl.Bsethome , 
    bSetPosition:=SR70_Vert_servo_ctrl.Bsetpos , 
	bMoveAbsolute:=SR70_Vert_servo_ctrl.ABSmove_Start , 
	bMoveRelative:=SR70_Vert_servo_ctrl.RELmove_Start , 
	bMoveTorque :=SR70_Vert_servo_ctrl.Torque_mode_Start,
	stManualModeAxis:=SR70_Vert_servo_status , 
	sAxisState=>SR70_Vert_servo_ctrl.Axis_State , 
	bAxis_ready=>SR70_Vert_servo_ctrl.Axis_ready , 
	bAxisInPosition=> SR70_Vert_servo_ctrl.Axis_In_Pos, 
	bAxisError=>SR70_Vert_servo_ctrl.Axis_Error , 
	bAxisEnabled=> SR70_Vert_servo_ctrl.Axis_Enabled, 
	bAxisHomed=> SR70_Vert_servo_ctrl.Axis_reference,
	bTorqueReached=> SR70_Vert_servo_ctrl.Trq_reached, 
	bSetPositionDone=>   ,
	bsafe_to_move=> ,
	bABS_Pos_done=> SR70_Vert_servo_ctrl.pos_done , 
	bHaltDone=> , 
	bSTOPDone=> , 
	bHomeDone=> , 
	bDone=> );	

OP70_GVL.SR70_HORI_servo(
	bAxis1_Ref_Switch:= temp, 
	bInit:= , 
	bErrorReset:=OP70_HMI_Reset OR Servo_Reset , 
	bEnable:= Servo_Enable, 
	bMoveVelocity:= , 
	bHalt:= , 
	bManualMode:= OP70_ManualSelected AND MANUAL_SELECTED,
	fHomePos:= , 
	fOverride:= , 
	fTargetPosition:= SR70_HORI_servo_ctrl.Position , 
	fTargetVelocity:= SR70_HORI_servo_ctrl.Velocity, 
	fAcc:= , 
	fDec:= ,
	Servo_High_Limit:= OP70_HMI_Hori_High_Limit,	
	Servo_Low_Limit:= OP70_HMI_Hori_Low_Limit,	 	
	WARNING_LIMIT:=1,	
	Actual_Torque=> SR70_HORI_servo_ctrl.Actual_Torque ,
	Actual_position=>SR70_HORI_servo_ctrl.Actual_Position ,
    Actual_velocity=>SR70_HORI_servo_ctrl.Actual_Velocity ,	
	bmove_home:=SR70_HORI_servo_ctrl.Axis_Home_Cmd ,
	baxis_in_home_pos=>SR70_HORI_servo_ctrl.Axis_In_Home ,
	Safe_move_Conditions:=Servo_Safety,
	Axis:= SR70_HORI_servo_Axis , 
	HME_WRITE_ADD:= 16#500B,	
	bHome:=SR70_HORI_servo_ctrl.Bsethome , 
    bSetPosition:=SR70_HORI_servo_ctrl.Bsetpos , 
	bMoveAbsolute:=SR70_HORI_servo_ctrl.ABSmove_Start , 
	bMoveRelative:=SR70_HORI_servo_ctrl.RELmove_Start , 
	bMoveTorque :=SR70_HORI_servo_ctrl.Torque_mode_Start,
	stManualModeAxis:=SR70_HORI_servo_status , 
	sAxisState=>SR70_HORI_servo_ctrl.Axis_State , 
	bAxis_ready=>SR70_HORI_servo_ctrl.Axis_ready , 
	bAxisInPosition=> SR70_HORI_servo_ctrl.Axis_In_Pos, 
	bAxisError=>SR70_HORI_servo_ctrl.Axis_Error , 
	bAxisEnabled=> SR70_HORI_servo_ctrl.Axis_Enabled, 
	bAxisHomed=> SR70_HORI_servo_ctrl.Axis_reference,
	bTorqueReached=> SR70_HORI_servo_ctrl.Trq_reached, 
	bSetPositionDone=>   ,
	bsafe_to_move=> ,
	bABS_Pos_done=> SR70_HORI_servo_ctrl.pos_done , 
	bHaltDone=> , 
	bSTOPDone=> , 
	bHomeDone=> , 
	bDone=> );

OP70_GVL.SR70_CONV_servo(
	bAxis1_Ref_Switch:= temp, 
	bInit:= , 
	bErrorReset:=OP70_HMI_Reset OR Servo_Reset , 
	bEnable:=Servo_Enable, 
	bMoveVelocity:=SR70_CONV_servo_ctrl.VELmove_Start , 
	bHalt:= , 
	bManualMode:= OP70_ManualSelected AND MANUAL_SELECTED ,
	fHomePos:= , 
	fOverride:= , 
	fTargetPosition:= SR70_CONV_servo_ctrl.Position, 
	fTargetVelocity:= SR70_CONV_servo_ctrl.Velocity, 
	LIMIT_BYPASS:=1,
	fAcc:= , 
	fDec:= ,
	Actual_Torque=> SR70_CONV_servo_ctrl.Actual_Torque ,
	Actual_position=>SR70_CONV_servo_ctrl.Actual_Position ,
    Actual_velocity=>SR70_CONV_servo_ctrl.Actual_Velocity ,	
	bmove_home:=SR70_CONV_servo_ctrl.Axis_Home_Cmd ,
	baxis_in_home_pos=>SR70_CONV_servo_ctrl.Axis_In_Home ,
	Safe_move_Conditions:=Servo_Safety,
	Axis:= SR70_CONV_servo_Axis , 
	HME_WRITE_ADD:= 16#500D,	
	bHome:=SR70_CONV_servo_ctrl.Bsethome , 
    bSetPosition:=SR70_CONV_servo_ctrl.Bsetpos , 
	bMoveAbsolute:=SR70_CONV_servo_ctrl.ABSmove_Start , 
	bMoveRelative:=SR70_CONV_servo_ctrl.RELmove_Start , 
	bMoveTorque :=SR70_CONV_servo_ctrl.Torque_mode_Start,
	stManualModeAxis:=SR70_CONV_servo_status , 
	sAxisState=>SR70_CONV_servo_ctrl.Axis_State , 
	bAxis_ready=>SR70_CONV_servo_ctrl.Axis_ready , 
	bAxisInPosition=> SR70_CONV_servo_ctrl.Axis_In_Pos, 
	bAxisError=>SR70_CONV_servo_ctrl.Axis_Error , 
	bAxisEnabled=> SR70_CONV_servo_ctrl.Axis_Enabled, 
	bAxisHomed=> SR70_CONV_servo_ctrl.Axis_reference,
	bTorqueReached=> SR70_CONV_servo_ctrl.Trq_reached, 
	bSetPositionDone=>   ,
	bsafe_to_move=>SR70_CONV_servo_ctrl.Safe_To_Move ,
	bABS_Pos_done=> SR70_CONV_servo_ctrl.pos_done , 
	bHaltDone=> , 
	bSTOPDone=> , 
	bHomeDone=> , 
	bDone=> );	
	
IF OP70_ManualSelected AND MANUAL_SELECTED THEN
	SR70_Vert_servo_status.targetVelocity:=50;
	SR70_Hori_servo_status.targetVelocity:=50;
	//SR70_CONV_servo_status.targetVelocity:=100;
	OP70_Gripper_LH_Gripper_ctrl.Velocity       :=  300;
	OP70_Gripper_RH_Gripper_ctrl.Velocity       :=  300;	
	OP70_Gripper_LH_Gripper_ctrl.ABSmove_Start:=LH_Gripper_bMove;
	OP70_Gripper_RH_Gripper_ctrl.ABSmove_Start:=RH_Gripper_bMove;
END_IF

//LH Rejection Cylinder
//move ZERO to STATUS
//CR70_LH_Rej_Cyl_Status:=0;

//Reset Auto Cmd IN Manual Mode & Homing
IF (OP70_Auto OR OP70_HomeRunning) THEN
	CR70_LH_Rej_Cyl.AutoCmd1:=FALSE;
	CR70_LH_Rej_Cyl.AutoCmd2:=FALSE;		
END_IF

// Safe Home
IF (TRUE) AND  (TRUE) THEN 
	CR70_LH_Rej_Cyl.SafeHome:= TRUE ;
ELSE 
	CR70_LH_Rej_Cyl.SafeHome:= FALSE ;
END_IF
// Safe Work
IF (TRUE) OR (TRUE) THEN 
	CR70_LH_Rej_Cyl.Safework:= TRUE ;
ELSE 
	CR70_LH_Rej_Cyl.Safework:= FALSE ;
END_IF
	
// Manual PB  Cyl Mapping
IF (OP70_HMI_LH_Rej_Cyl_Home_PB=TRUE) THEN
	CR70_LH_Rej_Cyl.ManualPB1:=TRUE;
ELSE 
	CR70_LH_Rej_Cyl.ManualPB1:=FALSE;
END_IF
	
IF (OP70_HMI_LH_Rej_Cyl_Work_PB=TRUE) THEN
	CR70_LH_Rej_Cyl.ManualPB2:=TRUE;
ELSE 
	CR70_LH_Rej_Cyl.ManualPB2:=FALSE;
END_IF
	
CR70_LH_Rej_Cyl(
	Auto:= OP70_AutoSelected , 
	Manual:= OP70_ManualSelected AND MANUAL_SELECTED, 
	ErrorActive:= , 
	ResetPB:= OP70_HMI_Reset, 
	Sensor1:= I70_LH_REJ_CYL_FWD_I1110_4, 
	Sensor2:= I70_LH_REJ_CYL_REV_I1110_5 , 
	ManualPB1:= , 
	ManualPB2:= , 
	AutoCmd1:= , 
	AutoCmd2:= , 
	OperationEnable:= OperationEnable , 
	SafeHome:= , 
	SafeWork:= , 
	HomingCmd1:= , 
	Pulse_1Sec:= Pulse_Block.Q1Hz , 
	BlinkingBit:= , 
	TimeOut1:=5 , 
	TimeOut2:=5 , 
	TimeOut3:=5 ,  
	Solenoid1=> O70_LH_REJ_CYL_FWD_Q1152_5  , 
	Solenoid2=> O70_LH_REJ_CYL_REV_Q1152_4 ,
	AlarmSensor1=> , 
	AlarmSensor2=> , 
	AlarmSolenoid1=> , 
	AlarmSolenoid2=> , 
	AllSignal=> , 
	AlarmPresent=> , 
	Position1=> , 
	Position2=> , 
	HomeSensorBlink=> , 
	WorkSensorBlink=> , 
	Status:=CR70_LH_Rej_Cyl_status );


//RH Rejection Cylinder
//move ZERO to STATUS
//CR70_RH_Rej_Cyl_Status:=0;

//Reset Auto Cmd IN Manual Mode & Homing
IF (OP70_Auto OR OP70_HomeRunning) THEN
	CR70_RH_Rej_Cyl.AutoCmd1:=FALSE;
	CR70_RH_Rej_Cyl.AutoCmd2:=FALSE;		
END_IF

// Safe Home
IF (TRUE) AND  (TRUE) THEN 
	CR70_RH_Rej_Cyl.SafeHome:= TRUE ;
ELSE 
	CR70_RH_Rej_Cyl.SafeHome:= FALSE ;
END_IF
// Safe Work
IF (TRUE) OR (TRUE) THEN 
	CR70_RH_Rej_Cyl.Safework:= TRUE ;
ELSE 
	CR70_RH_Rej_Cyl.Safework:= FALSE ;
END_IF
	
// Manual PB  Cyl Mapping
IF (OP70_HMI_RH_Rej_Cyl_Home_PB=TRUE) THEN
	CR70_RH_Rej_Cyl.ManualPB1:=TRUE;
ELSE 
	CR70_RH_Rej_Cyl.ManualPB1:=FALSE;
END_IF
	
IF (OP70_HMI_RH_Rej_Cyl_Work_PB=TRUE) THEN
	CR70_RH_Rej_Cyl.ManualPB2:=TRUE;
ELSE 
	CR70_RH_Rej_Cyl.ManualPB2:=FALSE;
END_IF
	
CR70_RH_Rej_Cyl(
	Auto:= OP70_AutoSelected ,  
	Manual:= OP70_ManualSelected AND MANUAL_SELECTED, 
	ErrorActive:= , 
	ResetPB:= OP70_HMI_Reset,                    
	Sensor1:= I70_RH_REJ_CYL_FWD_I1110_6, 
	Sensor2:= I70_RH_REJ_CYL_REV_I1110_7, 
	ManualPB1:= , 
	ManualPB2:= , 
	AutoCmd1:= , 
	AutoCmd2:= , 
	OperationEnable:=OperationEnable , 
	SafeHome:= , 
	SafeWork:= , 
	HomingCmd1:= , 
	Pulse_1Sec:= Pulse_Block.Q1Hz , 
	BlinkingBit:= , 
	TimeOut1:=5 , 
	TimeOut2:=5 , 
	TimeOut3:=5 , 
	Solenoid1=> O70_RH_REJ_CYL_FWD_Q1152_7 , 
	Solenoid2=> O70_RH_REJ_CYL_REV_Q1152_6 , 
	AlarmSensor1=> , 
	AlarmSensor2=> , 
	AlarmSolenoid1=>, 
	AlarmSolenoid2=> , 
	AllSignal=> , 
	AlarmPresent=> , 
	Position1=> , 
	Position2=> , 
	HomeSensorBlink=> , 
	WorkSensorBlink=> , 
	Status:=CR70_RH_Rej_Cyl_status );	

OP70_Gripper_LH_Gripper_ctrl.Velocity       :=  500;
OP70_Gripper_RH_Gripper_ctrl.Velocity       :=  500;	
OP70_Gripper_Current        :=  2;
OP70_Gripper_Acceleration   :=  2500;	
OP70_Gripper_Jerk           :=  50000;
	
OP70_Gripper_LH(
	iHW:= HwIn3 , 
	o_b_enable=> OP70_Gripper_LH_Gripper_ctrl.Axis_Enabled ,
	i_b_moveToPosition:=OP70_Gripper_LH_Gripper_ctrl.ABSmove_Start , 
	i_b_moveRelativ:= , 
	i_b_reference:=OP70_Gripper_LH_Gripper_ctrl.Reference_Start , 
	i_b_ackError:=OP70_HMI_Reset OR HMI_Reset, 
	i_u_targetPos:=OP70_Gripper_LH_Gripper_ctrl.Position , 
	i_u_targetVelocity:=OP70_Gripper_LH_Gripper_ctrl.Velocity , 
	i_u_targetCurrent:= OP70_Gripper_Current , 
	i_u_targetAcceleration:= OP70_Gripper_Acceleration , 
	i_u_targetJerk:= OP70_Gripper_Jerk , 
	i_b_ManualMode:= , 
	stManualModeAxis:=OP70_Gripper_LH_Manual_Axis , 
	Status=>OP70_Gripper_LH_Gripper_ctrl.Axis_State , 
	o_b_referenced=>OP70_Gripper_LH_Gripper_ctrl.Axis_reference , 
	o_b_reachedPos=> OP70_Gripper_LH_Gripper_ctrl.pos_done , 
	o_u_actualPosition=> OP70_Gripper_LH_Gripper_ctrl.Actual_Position , 
	o_b_error=> OP70_Gripper_LH_Gripper_ctrl.Axis_Error, 
	oHW=> HwOut3 );	
	
OP70_Gripper_RH(
	iHW:= HwIn4 , 
	o_b_enable => OP70_Gripper_RH_Gripper_ctrl.Axis_Enabled ,
	i_b_moveToPosition:=OP70_Gripper_RH_Gripper_ctrl.ABSmove_Start , 
	i_b_moveRelativ:= , 
	i_b_reference:=OP70_Gripper_RH_Gripper_ctrl.Reference_Start , 
	i_b_ackError:=OP70_HMI_Reset OR HMI_Reset, 
	i_u_targetPos:=OP70_Gripper_RH_Gripper_ctrl.Position , 
	i_u_targetVelocity:=OP70_Gripper_RH_Gripper_ctrl.Velocity , 
	i_u_targetCurrent:= OP70_Gripper_Current , 
	i_u_targetAcceleration:= OP70_Gripper_Acceleration , 
	i_u_targetJerk:= OP70_Gripper_Jerk , 
	i_b_ManualMode:= , 
	stManualModeAxis:=OP70_Gripper_RH_Manual_Axis , 
	Status=>OP70_Gripper_RH_Gripper_ctrl.Axis_State , 
	o_b_referenced=>OP70_Gripper_RH_Gripper_ctrl.Axis_reference , 
	o_b_reachedPos=> OP70_Gripper_RH_Gripper_ctrl.pos_done , 
	o_u_actualPosition=> OP70_Gripper_RH_Gripper_ctrl.Actual_Position , 
	o_b_error=> OP70_Gripper_RH_Gripper_ctrl.Axis_Error, 
	oHW=> HwOut4 );		
	
IF OP70_Gripper_LH_Gripper_ctrl.Axis_reference AND OP70_Gripper_LH_Open THEN
	OP70_Gripper_LH_Gripper_ctrl.Position:=OP70_Gripper_Wrk_POS;
	OP70_Gripper_LH_Gripper_ctrl.ABSmove_Start:=TRUE;
	IF OP70_Gripper_LH_Gripper_ctrl.pos_done AND In_range(OP70_Gripper_LH_Gripper_ctrl.Actual_Position,OP70_Gripper_Wrk_POS,1) THEN
		OP70_Gripper_LH_Open:=FALSE;
		OP70_Gripper_LH_Gripper_ctrl.ABSmove_Start:=0;	
		OP70_Gripper_LH_State:=1;
	END_IF
END_IF

IF OP70_Gripper_LH_Gripper_ctrl.Axis_reference AND OP70_Gripper_LH_Close THEN
	OP70_Gripper_LH_Gripper_ctrl.Position:=0.5;
	OP70_Gripper_LH_Gripper_ctrl.ABSmove_Start:=TRUE;
	IF OP70_Gripper_LH_Gripper_ctrl.pos_done AND In_range(OP70_Gripper_LH_Gripper_ctrl.Actual_Position,0,1) THEN
		OP70_Gripper_LH_Close:=FALSE;
		OP70_Gripper_LH_Gripper_ctrl.ABSmove_Start:=0;
		OP70_Gripper_LH_State:=0;
	END_IF
END_IF

IF  OP70_Gripper_RH_Gripper_ctrl.Axis_reference AND OP70_Gripper_RH_Open THEN
	OP70_Gripper_RH_Gripper_ctrl.Position:=OP70_Gripper_Wrk_POS;
	OP70_Gripper_RH_Gripper_ctrl.ABSmove_Start:=TRUE;
	IF OP70_Gripper_RH_Gripper_ctrl.pos_done AND In_range(OP70_Gripper_RH_Gripper_ctrl.Actual_Position,OP70_Gripper_Wrk_POS,1) THEN
		OP70_Gripper_RH_Open:=FALSE;
		OP70_Gripper_RH_Gripper_ctrl.ABSmove_Start:=0;
		OP70_Gripper_RH_State:=1;
	END_IF
END_IF

IF  OP70_Gripper_RH_Gripper_ctrl.Axis_reference AND OP70_Gripper_RH_Close THEN
	OP70_Gripper_RH_Gripper_ctrl.Position:=0.5;
	OP70_Gripper_RH_Gripper_ctrl.ABSmove_Start:=TRUE;
	IF OP70_Gripper_RH_Gripper_ctrl.pos_done AND In_range(OP70_Gripper_RH_Gripper_ctrl.Actual_Position,0,1) THEN
		OP70_Gripper_RH_Close:=FALSE;
		OP70_Gripper_RH_Gripper_ctrl.ABSmove_Start:=0;
		OP70_Gripper_RH_State:=0;
	END_IF	
END_IF

CASE Grip_Test OF
	1: OP70_Gripper_LH_Open:=1;
	   OP70_Gripper_RH_Open:=1;
	   Grip_Test:=2;
	   
	2: IF Test.Q THEN
		OP70_Gripper_LH_Close:=1;
		OP70_Gripper_RH_Close:=1;
			   Grip_Test:=1;
	   END_IF

END_CASE

Test(IN:= OP70_Gripper_RH_State AND OP70_Gripper_LH_State , PT:=T#500MS);	
	
	
(*OP70_GIUDE_GRP(														// FESTO GUIDE GRIPPER
	bAxis1_Ref_Switch:= , 
	bInit:=  , 
	bErrorReset:= Servo_Reset  , 
	bEnable:= Servo_Enable , /// MACHINE ERR REGISTER CHANGE
	bMoveVelocity:= , 
	bHalt:= , 
	bManualMode:= OP70_ManualSelected AND MANUAL_SELECTED , 									//MANUAL REGISTER CHANGE
	fHomePos:= , 
	fOverride:= , 
	fTargetPosition:= OP70_GIUDE_GRP_ctrl.Position, 
	fTargetVelocity:= OP70_GIUDE_GRP_ctrl.Velocity, 
	fAcc:= , 
	fDec:= , 
	Servo_High_Limit:= 100,	
	Servo_Low_Limit:= -100,	 	
	WARNING_LIMIT:=1,	
	Safe_move_Conditions:= Servo_Safety , // CHANGE
	Axis:= SR70_GUIDE_GRP_AXIS,
	bHome:=SR70_HORI_servo_ctrl.Bsethome , 
	bmove_home:=SR70_HORI_servo_ctrl.Axis_Home_Cmd ,
	bSetPosition:= FESTO_NOT_NEED , 
	bMoveAbsolute:= OP70_GIUDE_GRP_ctrl.ABSmove_Start, 
	bMoveRelative:= NOT_REQ , 
	bMoveTorque:= NOT_REQ , 
	stManualModeAxis:= OP70_GIUDE_GRP_Manual_Axis, 
 	sAxisState=> OP70_GIUDE_GRP_ctrl.Axis_State, 
	bAxis_ready=> , 
	bAxisInPosition=> , 
	bAxisError=> , 
	bAxisEnabled=> , 
	bAxisHomed=> , 
	bSetPositionDone=> , 
	bHaltDone=> , 
	bSTOPDone=> , 
	bHomeDone=> , 
	bDone=> , 
	bTorqueReached=> , 
	bsafe_to_move=> , 
	baxis_in_home_pos=> , 
	bABS_Pos_done=> OP70_GIUDE_GRP_ctrl.Axis_In_Pos, 
	Actual_position=>OP70_GIUDE_GRP_ctrl.Actual_Position,
	Actual_velocity=>OP70_GIUDE_GRP_ctrl.Actual_Velocity , 
	Actual_Torque=> );*)
IF OP70_ManualSelected AND MANUAL_SELECTED THEN	
	OP70_GIUDE_GRP_Manual_Axis.targetVelocity:=50;	
END_IF

OP70_GUIDE_GRP(
	bAxis1_Ref_Switch:= , 
	bInit:= , 
	bErrorReset:= Servo_Reset, 
	bEnable:= Servo_Enable, 
	bMoveVelocity:= , 
	bHalt:= , 
	bManualMode:= OP70_ManualSelected AND MANUAL_SELECTED , 
	bmove_home:= , 
	fHomePos:= , 
	fOverride:= , 
	fTargetPosition:=OP70_GIUDE_GRP_ctrl.Position , 
	fTargetVelocity:=OP70_GIUDE_GRP_ctrl.Velocity , 
	fAcc:= , 
	fDec:= , 
	Servo_High_Limit:=100 , 
	Servo_Low_Limit:= -100, 
	WARNING_LIMIT:= , 
	Safe_move_Conditions:= Servo_Safety,
	TORQUE_APPLIED := , 
	LIMIT_BYPASS:= , 
	Axis:= SR70_GUIDE_GRP_AXIS, 
	bHome:=OP70_GIUDE_GRP_ctrl.Bsethome, 
	bSetPosition:= FESTO_NOT_NEED, 
	bMoveAbsolute:= OP70_GIUDE_GRP_ctrl.ABSmove_Start, 
	bMoveRelative:= NOT_REQ, 
	bMoveTorque:= NOT_REQ, 
	stManualModeAxis:= OP70_GIUDE_GRP_Manual_Axis, 
	sAxisState=> OP70_GIUDE_GRP_ctrl.Axis_State, 
	baxis_in_home_pos=>OP70_GIUDE_GRP_ctrl.Axis_In_Home ,
	bAxis_ready=> , 
	bAxisInPosition=> , 
	bAxisError=> , 
	bAxisEnabled=> , 
	bAxisHomed=> , 
	bSetPositionDone=> , 
	bHaltDone=> , 
	bSTOPDone=> , 
	bHomeDone=> OP70_GIUDE_GRP_ctrl.Axis_Home_Done, 
	bDone=> , 
	bTorqueReached=> , 
	bsafe_to_move=> , 
	baxis_in_home_pos=> , 
	bABS_Pos_done=> OP70_GIUDE_GRP_ctrl.Axis_In_Pos, 
	Actual_position=> OP70_GIUDE_GRP_ctrl.Actual_Position, 
	Actual_velocity=>OP70_GIUDE_GRP_ctrl.Actual_Velocity , 
	Actual_Torque=> , 
	SERVO_LIMIT_WARNING=> );

END_PROGRAM

// ---- POUs/Programs/OP70/OP70_AUTOSEQUENCE.TcPOU
PROGRAM OP70_AUTOSEQUENCE
VAR
	OP70_Oring_OK 	: BOOL;
	FIXTURE_LH		: INT;
	FIXTURE_RH 		: INT;
	del : ton;
	tmp :BOOL;	
	Gripper_Delay: TON;
	Gripper_Aft_Place_Delay	: TON;
	Dry_Run : BOOL;
	OP70_STN_MOVER: INT;
	OP70_Cycle_Time_FB : FB_Cycletime;
	PAP_CYC_VAR : BOOL;
	OP70_PAP_Cycle_time : UDINT;
	OP70_Overall_Cyc_Time	: UDINT;
	OP70_PAP_Cycle_Time_FB : FB_Cycletime;
	OP70_Continous_Run : BOOL;
END_VAR

VAR PERSISTENT

END_VAR

// AUTO MODE
IF (NOT OP70_AutoSelected OR  OP70_ErrorActive OR OP70_HomeRunning ) THEN
	OP70_AutoRunning:= FALSE;
	OP70_Conveyor_ON:=FALSE;
	OP70_AutoSeq:= 10;
END_IF	

IF OP70_AutoSelected THEN
	OP70_GIUDE_GRP_ctrl.Position:=OP70_Guide_Pos;
	OP70_GIUDE_GRP_ctrl.Velocity:=50;	
	SR70_Vert_servo_ctrl.Velocity:=OP70_HMI_Servo_Speed_Vertical;
	SR70_HORI_servo_ctrl.Velocity:=OP70_HMI_Servo_Speed_Horizontal;	
END_IF

IF NOT OP70_AutoRunning THEN
    OP70_GIUDE_GRP_ctrl.Position:=0;
	OP70_GIUDE_GRP_ctrl.Velocity:=70;
	IF NOT In_Range(OP70_GIUDE_GRP_ctrl.Actual_Position,0,0.5) THEN
		OP70_GIUDE_GRP_ctrl.ABSmove_Start:=TRUE;
	END_IF	
END_IF

CASE OP70_AutoSeq OF
	    10: IF (OP70_AutoSelected) THEN		// Check Automode Selected
				OP70_AutoSeq:=20;
	        END_IF
		
	    20:IF ( NOT OP70_ErrorActive) THEN		//Check No error
		       OP70_AutoSeq:=30;
      	   END_IF
		   
      	30:IF (NOT OP70_HomeRunning) THEN		//Check No Homerunning
      		   OP70_AutoSeq :=40;
      	   END_IF
		   
        40:IF (OP70_Main.OP70_Modeselection_FB.TempHomeOK)THEN	//Check Machine in Home
      		   OP70_AutoSeq:= 50;
      	   END_IF
		   
      	50:IF ( NOT OP70_OperationCompleted) THEN		// Check Operation Completed Reset
      		   OP70_AutoSeq:=60;
      	   END_IF
		   
		60:IF  ( OP70_AutoRunning OR (NOT OP70_AutoRunning AND OP70_HMI_Cycle_Start )) THEN		//Machine Start in Fully Automatic or Press Cycle Start For Semi Automatic
		    OP70_GVL.OP70_HomeConditionOK:=TRUE;
	 			IF( OP70_Main.OP70_Modeselection_FB.HomeConditionOK AND OP70_AutoSelected) THEN
					OP70_GVL.OP70_AutoRunning:=TRUE;
					OP70_GVL.OP70_StepRunning:= FALSE;				
				ELSIF (OP70_Main.OP70_Modeselection_FB.HomeConditionOK AND OP70_StepSelected) THEN
					OP70_GVL.OP70_AutoRunning:=FALSE;
					OP70_GVL.OP70_StepRunning:= TRUE;
				END_IF;
		  END_IF
		   IF ((OP70_AutoRunning OR OP70_StepRunning) AND OP70_StartEnable) THEN
			   	OP70_GIUDE_GRP_ctrl.ABSmove_Start:=TRUE;
				OP70_Conveyor_ON:=TRUE;
				OP70_AutoSeq:= 65;
		   END_IF	
		   
		65 :  OP70_Gripper_LH_Close:=TRUE;  //CHECKING GRIPPER STATE BEFORE GRIPPING
			  OP70_Gripper_RH_Close:=TRUE;
			  IF NOT OP70_Gripper_LH_State AND NOT OP70_Gripper_RH_State THEN
				   OP70_AutoSeq:=66;
			  ELSE 	   
				   OP70_AutoSeq:=220;
			  END_IF 
			  
	    66: PAP_CYC_VAR:=1;
			IF OP70_pick_ready THEN
				OP70_AutoSeq:=70;
			ELSE 
				OP70_AutoSeq:=86;	
			END_IF 
		   
		70 : //MOVING HORIZONTAL SERVO TO PICK POSITION
			  IF (OP70_HORI_SERVO_ON_SFE_WRK_PICK OR OP70_HORI_SERVO_ON_SFE_WRK OR OP70_HORI_SERVO_ON_HOME OR OP70_HORI_SERVO_ON_WRK_PLACE OR OP70_HORI_SERVO_ON_WRK_PICK )AND OP70_HORI_SERVO_POS_DONE AND NOT SR70_HORI_servo_ctrl.ABSmove_Start THEN 
			   SR70_Hori_servo_ctrl.Position:=OP70_HORI_SERVO_PICK_POS;
               OP70_AutoSeq:=80; 			  
	          END_IF
			 
		80 :  SR70_HORI_servo_ctrl.ABSmove_Start := TRUE;     //HORIZONTAL SERVO MOVING
		       IF OP70_HORI_SERVO_ON_WRK_PICK THEN
				   SR70_HORI_servo_ctrl.ABSmove_Start := FALSE;
				   IF OP70_Gripper_LH_State AND OP70_Gripper_RH_State THEN
				        OP70_AutoSeq:=85;
				   ELSE 
						OP70_AutoSeq:=82;
				   END_IF
			   END_IF
		
	  	82 :  OP70_Gripper_LH_Close:=TRUE;  //CHECKING GRIPPER STATE BEFORE GRIPPING
			  OP70_Gripper_RH_Close:=TRUE;
			  IF NOT OP70_Gripper_LH_State AND NOT OP70_Gripper_RH_State THEN
				   OP70_AutoSeq:=85;
			  END_IF
			   
		85:	   // MOVING VERTICAL SERVO TO PICK POSITION
               IF  OP70_HORI_SERVO_ON_WRK_PICK AND (OP70_VERT_SERVO_ON_SFE_WRK OR OP70_VERT_SERVO_ON_HOME) AND 
				   OP70_VERT_SERVO_POS_DONE AND NOT SR70_VERT_servo_ctrl.ABSmove_Start  THEN
				   SR70_Vert_servo_ctrl.Position:=OP70_VERT_SERVO_PICK_POS;
				   SR70_VERT_servo_ctrl.ABSmove_Start := TRUE;
              	   OP70_AutoSeq:=100;			   
			   END_IF

	    86:   IF (OP70_HORI_SERVO_ON_SFE_WRK OR OP70_HORI_SERVO_ON_HOME OR OP70_HORI_SERVO_ON_WRK_PLACE OR OP70_HORI_SERVO_ON_WRK_PICK )AND OP70_HORI_SERVO_POS_DONE AND NOT SR70_HORI_servo_ctrl.ABSmove_Start THEN 
			    SR70_Hori_servo_ctrl.Position:=OP70_HORI_SERVO_SAFE_PICK_POS;
			    SR70_HORI_servo_ctrl.ABSmove_Start := TRUE;
                OP70_AutoSeq:=90;
			  END_IF
			   		  
		90 :  IF OP70_pick_ready THEN  // WAITING FOR O-RING TO BE OK AND THEN MOVING THE VERTICAL SERVO
			 		SR70_Hori_servo_ctrl.Position:=OP70_HORI_SERVO_PICK_POS;
					//SR70_Hori_servo_ctrl.ABSmove_Start := TRUE;
					OP70_AutoSeq:=92;
		      END_IF	
			  				
		92:  SR70_Hori_servo_ctrl.ABSmove_Start := TRUE;
			 IF OP70_HORI_SERVO_ON_WRK_PICK THEN
				 SR70_Vert_servo_ctrl.Position:=OP70_VERT_SERVO_PICK_POS;
				 SR70_VERT_servo_ctrl.ABSmove_Start := TRUE;
				 OP70_AutoSeq:=100;
			 END_IF 
	   
	   100 : IF OP70_VERT_SERVO_ON_WRK_PICK AND NOT SR70_VERT_servo_ctrl.ABSmove_Start THEN
				 SR70_VERT_servo_ctrl.ABSmove_Start := FALSE;
				 SR70_Vert_servo_ctrl.Position:=OP70_VERT_SERVO_SFE_WRK_POS; // FEEDING SAFE-WORK POSITION TO VERTICAL SERVO
              	 OP70_AutoSeq:=110;			   
			  END_IF	   
			 
      110:  IF NOT OP70_Grip_LH_Bypass THEN
				OP70_Gripper_LH_Open:=TRUE; 
			END_IF	
			IF NOT OP70_Grip_RH_Bypass THEN
    			OP70_Gripper_RH_Open:=TRUE;
			END_IF	
			IF Gripper_Delay.Q THEN
				 OP70_AutoSeq:=120;
		    END_IF
    		
      120: SR70_Hori_servo_ctrl.Position:=(OP70_HORI_SERVO_PICK_POS+OP70_Hori_Ser_Jerk_Pos);
	  	   SR70_HORI_servo_ctrl.ABSmove_Start := TRUE;
		   OP70_AutoSeq:=130;

    		   
      130:  SR70_HORI_servo_ctrl.ABSmove_Start := 0;
			SR70_VERT_servo_ctrl.ABSmove_Start := TRUE;	   //MOVING VERTICL SERVO TO SAFE-WORK
            IF OP70_VERT_SERVO_ON_SFE_WRK  THEN
    	      SR70_VERT_servo_ctrl.ABSmove_Start := FALSE;
			  OP70_pick_done:=TRUE;
              OP70_AutoSeq:=140;   
    		END_IF
    		   
      140:  IF (NOT OP70_Gripper_LH_State AND OP70_Grip_LH_Bypass ) AND OP70_Gripper_RH_State THEN  
    			OP70_AutoSeq:=150;
			ELSIF (NOT OP70_Gripper_RH_State AND OP70_Grip_RH_Bypass) AND OP70_Gripper_LH_State THEN
				OP70_AutoSeq:=150;
			ELSIF OP70_Gripper_LH_State AND OP70_Gripper_RH_State THEN  
    			OP70_AutoSeq:=150;
			ELSIF (NOT OP70_Gripper_LH_State AND NOT OP70_Grip_LH_Bypass) OR (NOT OP70_Gripper_RH_State AND NOT OP70_Grip_RH_Bypass) THEN	
				OP70_AutoSeq:=220;
			ELSIF OP70_Grip_LH_Bypass AND OP70_Grip_RH_Bypass THEN
				OP70_AutoSeq:=250;
			END_IF	
    	    		  
       150:  IF OP70_VERT_SERVO_ON_SFE_WRK  THEN // FEEDING PLACE POSITION TO HORIZONTAL SERVO
    		   SR70_Hori_servo_ctrl.Position:=OP70_HORI_SERVO_PLACE_POS;
               OP70_AutoSeq:=160;			 
    		 END_IF
    		   
       160:  SR70_HORI_servo_ctrl.ABSmove_Start := TRUE;    // MOVING HORIZONTAL SERVO TO PLACE POSITION
    		   IF OP70_HORI_SERVO_ON_WRK_PLACE THEN
    			 SR70_HORI_servo_ctrl.ABSmove_Start := FALSE;
    			 OP70_AutoSeq:=170;
    		   END_IF
       
       170: PAP_CYC_VAR:=0;
			IF OP70_HORI_SERVO_ON_WRK_PLACE AND NOT SR70_VERT_servo_ctrl.ABSmove_Start AND OP70_VERT_SERVO_ON_SFE_WRK AND OP70_STN_ENABLE THEN
    	   		SR70_Vert_servo_ctrl.Position:=OP70_VERT_SERVO_PLACE_POS;
              	OP70_AutoSeq:=175;	
      		END_IF
			
	   175: IF FIXTURE_LH<>60 AND FIXTURE_RH<>60 THEN
		   		OP70_AutoSeq:=250;	
			ELSIF FIXTURE_LH<>60 OR FIXTURE_RH<>60 THEN
				OP70_AutoSeq:=260;	
			ELSE
				OP70_AutoSeq:=180;		
	  	    END_IF			
    		
       180: SR70_VERT_servo_ctrl.ABSmove_Start := TRUE; //MOVING VERTICAL SERVO TO PLACE POSITION
    		IF OP70_VERT_SERVO_ON_WRK_PLACE THEN
    			SR70_VERT_servo_ctrl.ABSmove_Start := FALSE;
    			OP70_AutoSeq:=190;	
    		END_IF	
			
       190: IF FIXTURE_LH=60 AND NOT OP70_Grip_LH_Bypass THEN 
				OP70_Gripper_LH_Close:=TRUE;	
			END_IF	
			IF FIXTURE_RH=60 AND NOT OP70_Grip_RH_Bypass THEN 
				OP70_Gripper_RH_Close:=TRUE;	
			END_IF	
			tmp:=1;
			IF del.Q THEN		
				OP70_AutoSeq:=200;
			END_IF
			OP70_CURR_MOVER			:=OP70_STN_MOVER;
			
       200:  //MOVING BACK TO VERTICAL SERVO SAFE POSITION
    		 IF OP70_VERT_SERVO_ON_WRK_PLACE AND NOT SR70_VERT_servo_ctrl.ABSmove_Start THEN
    		   SR70_Vert_servo_ctrl.Position:=OP70_VERT_SERVO_SFE_WRK_POS;
               OP70_AutoSeq:=201;		   
    		 END_IF 

	   201: IF Dry_Run THEN
				OP70_AutoSeq:=210; 
			END_IF
			IF  FIXTURE_LH=60 AND FIXTURE_RH=60 THEN
				MOVER_CMP_STATUS[OP70_CURR_MOVER][1]:=70 ;
				MOVER_CMP_STATUS[OP70_CURR_MOVER][2]:=70 ;
				OP70_AutoSeq:=210;
			ELSIF FIXTURE_LH=60 THEN
				MOVER_CMP_STATUS[OP70_CURR_MOVER][1]:=70 ;
				OP70_AutoSeq:=210;
			ELSIF FIXTURE_RH=60 THEN
				MOVER_CMP_STATUS[OP70_CURR_MOVER][2]:=70 ;
				OP70_AutoSeq:=210;
			END_IF
    		 
       210:	 //PROCEEDING FOR NEXT CYCLE  
			  SR70_VERT_servo_ctrl.ABSmove_Start := TRUE;         
              IF OP70_VERT_SERVO_ON_SFE_WRK OR OP70_VERT_SERVO_ON_HOME  THEN
    			  SR70_VERT_servo_ctrl.ABSmove_Start := FALSE;
				  OP70_STN_ENABLE:=0;	  
    			  IF OP70_Gripper_LH_State OR OP70_Gripper_RH_State THEN
    		  		OP70_AutoSeq:=220;
    			  ELSIF (MOVER_CMP_STATUS[OP70_STN_MOVER][1]=70 OR MOVER_CMP_STATUS[OP70_STN_MOVER][2]=70) OR Dry_Run THEN
					STATION_DONE[OP70_CURR_MOVER][OP70_XTS_POS_NO]			:= TRUE;
					OP70_AutoSeq:=66;  
				  END_IF			  
    		  END_IF
    		  
       220:  IF (OP70_VERT_SERVO_ON_SFE_WRK OR OP70_VERT_SERVO_ON_HOME OR OP70_VERT_SERVO_ON_WRK_PLACE) AND NOT SR70_HORI_servo_ctrl.ABSmove_Start AND (OP70_HORI_SERVO_ON_WRK_PLACE OR OP70_HORI_SERVO_ON_WRK_Pick)  THEN
    		  SR70_Hori_servo_ctrl.Position:=OP70_HORI_SERVO_SFE_WRK_POS;
			  SR70_Vert_servo_ctrl.Position:=OP70_VERT_SERVO_SFE_WRK_POS;
			  SR70_VERT_servo_ctrl.ABSmove_Start := TRUE;
              OP70_AutoSeq:=240;			  
    		 END_IF  
    	
       240:  SR70_HORI_servo_ctrl.ABSmove_Start := TRUE;
             IF OP70_HORI_SERVO_ON_SFE_WRK THEN
    	  	   SR70_HORI_servo_ctrl.ABSmove_Start := FALSE;
      		   OP70_Gripper_RH_Close:=TRUE;	
    		   OP70_Gripper_LH_Close:=TRUE; 			   
      		 END_IF
    		 IF NOT OP70_Gripper_LH_State AND NOT OP70_Gripper_RH_State THEN
    		   OP70_AutoSeq:=66;
    		 END_IF
			 
		250://MOVER_CMP_STATUS[OP70_CURR_MOVER][1]:=71;
			//MOVER_CMP_STATUS[OP70_CURR_MOVER][2]:=71;
			OP70_STN_ENABLE:=0;	
			IF (MOVER_CMP_STATUS[OP70_STN_MOVER][1]=71 AND MOVER_CMP_STATUS[OP70_STN_MOVER][2]=71) THEN
				MOVER_STP_NO[OP70_CURR_MOVER]	:= (OP160_XTS_POS_NO*10);
			ELSE		
				STATION_DONE[OP70_CURR_MOVER][OP70_XTS_POS_NO]			:= TRUE;
			END_IF
				OP70_AutoSeq:=170; 	
	   260: SR70_Hori_servo_ctrl.Position:=OP70_HORI_SERVO_SFE_WRK_POS;
			SR70_Hori_servo_ctrl.ABSmove_Start:=TRUE;
			IF OP70_HORI_SERVO_ON_SFE_WRK THEN
				OP70_AutoSeq:=270; 
			END_IF
			
	   270: IF FIXTURE_LH<>60 AND NOT OP70_Grip_LH_Bypass THEN
				OP70_Gripper_LH_Close:=TRUE;
				IF NOT OP70_Gripper_LH_State THEN
					OP70_AutoSeq:=280; 
				END_IF
			ELSE
				OP70_AutoSeq:=280;	
			END_IF	
			
	   280: IF FIXTURE_RH<>60 AND NOT OP70_Grip_RH_Bypass THEN
				OP70_Gripper_RH_Close:=TRUE;
				IF NOT OP70_Gripper_RH_State THEN
					OP70_AutoSeq:=290; 
				END_IF
			ELSE
				OP70_AutoSeq:=290;	
			END_IF	

	   290: SR70_Hori_servo_ctrl.Position:=OP70_HORI_SERVO_PLACE_POS;
			SR70_Hori_servo_ctrl.ABSmove_Start:=TRUE;
			IF OP70_HORI_SERVO_ON_WRK_PLACE THEN
				OP70_AutoSeq:=180;	
			END_IF			 

END_CASE


OP70_STN_ENABLE:=OP70_Continous_Run;
				
OP70_Cycle_Time_FB(i_b_startTime:=OP70_STN_ENABLE , i_b_stopTime:= NOT OP70_STN_ENABLE , o_t_StationTime=>OP70_Cycle_time );					
OP70_PAP_Cycle_Time_FB(i_b_startTime:=PAP_CYC_VAR , i_b_stopTime:= NOT PAP_CYC_VAR , o_t_StationTime=>OP70_PAP_Cycle_time );					
OP70_Overall_Cyc_Time:=OP70_Cycle_time+OP70_PAP_Cycle_time;
	

Gripper_Delay(IN:=(OP70_AutoSeq=110),PT:=T#500MS);

Dry_Run:=All_Station_Dry_Run;
IF Dry_run THEN
	FIXTURE_LH :=60;	
    FIXTURE_RH :=60;
ELSE 
	FIXTURE_LH:=MOVER_CMP_STATUS[OP70_STN_MOVER][1];
	FIXTURE_RH:=MOVER_CMP_STATUS[OP70_STN_MOVER][2];	
END_IF	

del(IN:=tmp,PT:=T#700MS);
IF del.Q THEN
	tmp:=FALSE;
END_IF

// ################################			STATION ENABLE		####################################


OP70_STN_MOVER					:= MOVER_POSITION[OP70_XTS_POS_NO];

IF AUTO_WITH_XTS THEN
IF OP70_STN_MOVER>0 THEN
IF NOT(END_OF_CYCLE AND MOVER_CMP_STATUS[OP70_STN_MOVER][1]=5 AND MOVER_CMP_STATUS[OP70_STN_MOVER][2]=5)THEN	
	OP70_STN_ENABLE					:= MOVER_POS_RECHED[OP70_STN_MOVER] AND ((MOVER_CMP_STATUS[OP70_STN_MOVER][1]=60)OR
										(MOVER_CMP_STATUS[OP70_STN_MOVER][2]=60)) AND STATION_ENABLE_CONTROL;	
ELSE
	STATION_DONE[OP70_STN_MOVER][OP70_XTS_POS_NO]			:= TRUE;	
END_IF
ELSE
	OP70_STN_ENABLE					:= FALSE;
END_IF	
END_IF

END_PROGRAM

// ---- POUs/Programs/OP70/OP70_Camera_FB.TcPOU
PROGRAM OP70_Camera_FB
VAR
	OP70_LH_Camera 			        : FB_Cognex_ProfiNET_1;

	
	OP70_LH_Acquisition_Status AT %I*    :Acquisition_Status;
	OP70_LH_Inspection_Status  AT %I*    :Inspection_Status;	
	OP70_LH_Acquisition_ID     AT %I*    :UINT;
	OP70_LH_Inspection_ID   	 AT %I*  :UINT;
	OP70_LH_Error_code      	 AT %I*  :UINT;
	OP70_LH_Current_Job_ID  	 AT %I*  :UINT;
	OP70_LH_Result_code     	 AT %I*  :UINT;
	OP70_LH_Cam_Result      	 AT %I*  :ARRAY[0..63] OF BYTE;	
	OP70_LH_Acquisition_Control AT %Q*  : Acquisition_Control;
	OP70_LH_Inspection_Control  AT %Q*  : Inspection_Control;
	OP70_LH_Command_word		AT %Q*  : UINT;
	OP70_LH_Union                       : UNION_64Byte;

	OP70_RH_Camera 			          : FB_Cognex_ProfiNET_1;

	
	OP70_RH_Acquisition_Status AT %I*    :Acquisition_Status;
	OP70_RH_Inspection_Status  AT %I*    :Inspection_Status;	
	OP70_RH_Acquisition_ID     AT %I*    :UINT;
	OP70_RH_Inspection_ID   	 AT %I*  :UINT;
	OP70_RH_Error_code      	 AT %I*  :UINT;
	OP70_RH_Current_Job_ID  	 AT %I*  :UINT;
	OP70_RH_Result_code     	 AT %I*  :UINT;
	OP70_RH_Cam_Result      	 AT %I*  :ARRAY[0..63] OF BYTE;	
	OP70_RH_Acquisition_Control AT %Q*  : Acquisition_Control;
	OP70_RH_Inspection_Control  AT %Q*  : Inspection_Control;
	OP70_RH_Command_word		AT %Q*  : UINT;
	OP70_RH_Union                       : UNION_64Byte;
END_VAR


	OP70_LH_Camera (
	tTimeout:= , 
	sJob_Name:= , 
	camera_ready=> OP70_LH_Camera_Ready,
	Camera_online=> OP70_LH_Camera_Online,
	stCognex_record_status:=OP70_LH_Acquisition_Status, 
	Acquisition_ID:=OP70_LH_Acquisition_ID , 
	stCognex_Inspection_status:=OP70_LH_Inspection_Status, 
	Error_Code:=OP70_LH_Error_code , 
	wcommand_control_in:= OP70_LH_Current_Job_ID, 
	aResults_64_Bytes:= OP70_LH_Cam_Result, 
	number_of_inspections:=OP70_LH_Inspection_ID , 
	iresult_code:= OP70_LH_Result_code, 
	bTarget_job_ID:=OP70_LH_Target_Job_ID , 
	Error_Status_message=> OP70_LH_Error_status, 
	bError=> OP70_LH_Camera_Error, 
	stCognex_record_control=>OP70_LH_Acquisition_Control , 
	stCognex_inspection_control=>OP70_LH_Inspection_Control , 
	wCommandControl_out=>OP70_LH_Command_word , 
	aUser_data_64_Byte=> OP70_LH_Union.aArrayOfByte, 
	bJob_loading_completed=>OP70_LH_Job_Change_Complete , 
	bJob_load_failed=>OP70_LH_Job_Change_Error , 
	bInspection_Result_IO=>  , 
	bInspection_Result_NIO=> , 
	bTXTSM_Error_Job_Change=> OP70_LH_Job_Change_Error, 
	bPictureTakenComplete=> OP70_LH_Picture_Taken, 
	Loaded_Job_ID=>OP70_LH_Loaded_Job_ID	 , 
	bClear_Error:= HMI_Reset, 
	bJob_change_start:= OP70_LH_Camera_Job_Change_start, 
	TXTSM_camera_not_online=>OP70_LH_Camera_Error	 , 
	bTrigger_start:= OP70_LH_Camera_Trigger );
	
	OP70_RH_Camera (
	tTimeout:= , 
	sJob_Name:= , 
	camera_ready=> OP70_RH_Camera_Ready,
	Camera_online=> OP70_RH_Camera_Online,
	stCognex_record_status:=OP70_RH_Acquisition_Status, 
	Acquisition_ID:=OP70_RH_Acquisition_ID , 
	stCognex_Inspection_status:=OP70_RH_Inspection_Status, 
	Error_Code:=OP70_RH_Error_code , 
	wcommand_control_in:= OP70_RH_Current_Job_ID, 
	aResults_64_Bytes:= OP70_RH_Cam_Result, 
	number_of_inspections:=OP70_RH_Inspection_ID , 
	iresult_code:= OP70_RH_Result_code, 
	bTarget_job_ID:=OP70_RH_Target_Job_ID , 
	Error_Status_message=> OP70_RH_Error_status, 
	bError=> OP70_RH_Camera_Error, 
	stCognex_record_control=>OP70_RH_Acquisition_Control , 
	stCognex_inspection_control=>OP70_RH_Inspection_Control , 
	wCommandControl_out=>OP70_RH_Command_word , 
	aUser_data_64_Byte=> OP70_RH_Union.aArrayOfByte, 
	bJob_loading_completed=>OP70_RH_Job_Change_Complete , 
	bJob_load_failed=>OP70_RH_Job_Change_Error , 
	bInspection_Result_IO=>  , 
	bInspection_Result_NIO=> , 
	bTXTSM_Error_Job_Change=> OP70_RH_Job_Change_Error, 
	bPictureTakenComplete=> OP70_RH_Picture_Taken, 
	Loaded_Job_ID=>OP70_RH_Loaded_Job_ID	 , 
	bClear_Error:= HMI_Reset, 
	bJob_change_start:= OP70_RH_Camera_Job_Change_start, 
	TXTSM_camera_not_online=>OP70_RH_Camera_Error	 , 
	bTrigger_start:= OP70_RH_Camera_Trigger );

END_PROGRAM

// ---- POUs/Programs/OP70/OP70_Error.TcPOU
PROGRAM OP70_Error
VAR
	OP70_Step_Err_1: TON;
	OP70_Step_Err_2: TON;
	OP70_Step_Err_3: TON;
	OP70_Step_Err_4: TON;
	OP70_Step_Err_5: TON;
	OP70_Step_Err_6: TON;
END_VAR

// Set ERROR ACTIVE
IF ((OP70_GVL.OP70_ErrorWord_0<>0) OR (OP70_GVL.OP70_ErrorWord_1<>0) OR (OP70_GVL.OP70_ErrorWord_2<>0)) THEN
	OP70_GVL.OP70_ErrorActive:= TRUE;
END_IF

//Reset ErrorActive
IF (OP70_GVL.OP70_HMI_Reset) OR HMI_Reset THEN 
	OP70_GVL.OP70_ErrorActive:= FALSE;
	OP70_GVL.OP70_ErrorWord_0:= 0;
	OP70_GVL.OP70_ErrorWord_1:= 0;
	OP70_GVL.OP70_ErrorWord_2:= 0;	
END_IF

// Auto Seq Step Error

//Horizontal Servo is not in home or safe-work position 
OP70_Step_Err_1(IN:=(OP70_GVL.OP70_AutoSeq=70) , PT:=T#5S , Q=> , ET=> );
IF (OP70_GVL.OP70_AutoSeq=70 AND OP70_Step_Err_1.Q) THEN
	OP70_GVL.OP70_ErrorWord_0.0:=TRUE;
END_IF


//Horizontal Servo not reaching pick position 
OP70_Step_Err_1(IN:=(OP70_GVL.OP70_AutoSeq=80) , PT:=T#5S , Q=> , ET=> );
IF (OP70_GVL.OP70_AutoSeq=80 AND NOT OP70_HORI_SERVO_ON_WRK_PICK AND OP70_Step_Err_1.Q) THEN
	OP70_GVL.OP70_ErrorWord_0.1:=TRUE;
END_IF

// Gripper is not closing
OP70_Step_Err_2(IN:=OP70_GVL.OP70_AutoSeq=82 , PT:=T#5S , Q=> , ET=> );
IF (OP70_GVL.OP70_AutoSeq=82 AND OP70_Step_Err_2.Q) THEN
	OP70_GVL.OP70_ErrorWord_0.2:=TRUE;
END_IF

// Vertical Servo not reaching work position 
OP70_Step_Err_3(IN:=OP70_GVL.OP70_AutoSeq=100 , PT:=T#5S , Q=> , ET=> );
IF (OP70_GVL.OP70_AutoSeq=100 AND OP70_Step_Err_3.Q) THEN
	OP70_GVL.OP70_ErrorWord_0.3:=TRUE;
END_IF

// Vertical Servo not reaching safe-work position 
OP70_Step_Err_3(IN:=OP70_GVL.OP70_AutoSeq=170 , PT:=T#5S , Q=> , ET=> );
IF (OP70_GVL.OP70_AutoSeq=170 AND OP70_Step_Err_3.Q) THEN
	OP70_GVL.OP70_ErrorWord_0.4:=TRUE;
END_IF

// Checking the gripper condition is opened or not
OP70_Step_Err_3(IN:=OP70_GVL.OP70_AutoSeq=140 , PT:=T#5S , Q=> , ET=> );
IF (OP70_GVL.OP70_AutoSeq=140 AND OP70_Step_Err_3.Q) THEN
	OP70_GVL.OP70_ErrorWord_0.5:=TRUE;
END_IF

//  Horizontal sevo not moving to place position
OP70_Step_Err_3(IN:=OP70_GVL.OP70_AutoSeq=160 , PT:=T#5S , Q=> , ET=> );
IF (OP70_GVL.OP70_AutoSeq=160 AND OP70_Step_Err_3.Q) THEN
	OP70_GVL.OP70_ErrorWord_0.6:=TRUE;
END_IF

//  Vertical sevo not moving to place position
OP70_Step_Err_3(IN:=OP70_GVL.OP70_AutoSeq=180 , PT:=T#5S , Q=> , ET=> );
IF (OP70_GVL.OP70_AutoSeq=180 AND OP70_Step_Err_3.Q) THEN
	OP70_GVL.OP70_ErrorWord_0.7:=TRUE;
END_IF

// Vertical Servo not reaching safe-work position 
OP70_Step_Err_3(IN:=OP70_GVL.OP70_AutoSeq=210 , PT:=T#5S , Q=> , ET=> );
IF (OP70_GVL.OP70_AutoSeq=210 AND OP70_Step_Err_3.Q) THEN
	OP70_GVL.OP70_ErrorWord_0.8:=TRUE;
END_IF

//  Horizontal sevo not moving to safe work position
OP70_Step_Err_3(IN:=OP70_GVL.OP70_AutoSeq=240 , PT:=T#5S , Q=> , ET=> );
IF (OP70_GVL.OP70_AutoSeq=240 AND OP70_Step_Err_3.Q) THEN
	OP70_GVL.OP70_ErrorWord_0.9:=TRUE;
END_IF

END_PROGRAM

// ---- POUs/Programs/OP70/OP70_Initialize_Seq.TcPOU
PROGRAM OP70_Initialize_Seq
VAR
	Homing_Check_Timer : TON;
END_VAR

IF OP70_GIUDE_GRP_ctrl.Axis_In_Home AND OP70_GIUDE_GRP_ctrl.Axis_Home_Done AND(SR70_Vert_servo_ctrl.Axis_In_Home) AND OP70_HORI_SERVO_ON_HOME AND NOT OP70_Gripper_LH_State AND NOT OP70_Gripper_RH_State AND (OP70_Gripper_LH_Gripper_ctrl.Axis_reference OR OP70_Grip_LH_Bypass) AND (OP70_Gripper_RH_Gripper_ctrl.Axis_reference OR OP70_Grip_RH_Bypass) THEN
	OP70_Temp_hmeOK:=TRUE;
	OP70_HomeRunning:=FALSE;
	OP70_Homing_Seq:=0;
ELSE
	OP70_Temp_hmeOK:=FALSE;	
END_IF

CASE OP70_Homing_Seq OF
	0: IF (OP70_AutoSelected AND NOT OP70_HomeRunning AND NOT OP70_ErrorActive AND NOT OP70_AutoRunning AND NOT OP70_StepRunning AND NOT OP70_Temp_hmeOK) THEN
		OP70_HomeRunning:=TRUE;
		OP70_Homing_Seq:=10;	
	   END_IF
	   
	10:IF (OP70_HomeRunning AND (OP70_HMI_Homing) OR HMI_Reset)THEN 
		IF (SR70_Vert_servo_ctrl.Axis_In_Home) THEN 
			SR70_Vert_servo_ctrl.Axis_Home_Cmd:=FALSE;
		    OP70_Homing_Seq:=20;
		ELSE
			SR70_Vert_servo_ctrl.Position:=0;
			SR70_Vert_servo_ctrl.Velocity:=100;
			SR70_Vert_servo_ctrl.ABSmove_Start:=TRUE;
			SR70_Vert_servo_ctrl.Axis_Home_Cmd:=TRUE;		
	    END_IF
	   END_IF		
	   
   20: IF (OP70_HORI_SERVO_ON_HOME) THEN 	   
  			SR70_Hori_servo_ctrl.Axis_Home_Cmd:=FALSE;
		ELSE
			SR70_Hori_servo_ctrl.Position:=OP70_HORI_SERVO_HME_POS;
			SR70_Hori_servo_ctrl.Velocity:=100;
			SR70_Hori_servo_ctrl.ABSmove_Start:=TRUE;
	    END_IF
		OP70_Homing_Seq:=40;
		
   40: 	OP70_Gripper_LH_Gripper_ctrl.Reference_Start := Pulse_Block.Q2Hz;
   		IF  OP70_Gripper_LH_Gripper_ctrl.Axis_reference THEN
		  OP70_Gripper_LH_Close:=1;	
		  OP70_Gripper_LH_State:=0;
		  OP70_Homing_Seq:=50;
		END_IF
		
   50: 	OP70_Gripper_RH_Gripper_ctrl.Reference_Start := Pulse_Block.Q2Hz;
   		IF  OP70_Gripper_RH_Gripper_ctrl.Axis_reference THEN
			OP70_Gripper_RH_Close:=1;
   			OP70_Gripper_RH_State:=0;
			OP70_Homing_Seq:=60;
		END_IF	
		
   60: 	CR70_LH_Rej_Cyl.HomingCmd1:=TRUE;	
		IF CR70_LH_Rej_Cyl.Position1 THEN
			CR70_LH_Rej_Cyl.HomingCmd1:=FALSE;
			OP70_Homing_Seq:=70;
		END_IF
		
   70:	CR70_RH_Rej_Cyl.HomingCmd1:=TRUE;	
		IF CR70_RH_Rej_Cyl.Position1 THEN
			CR70_RH_Rej_Cyl.HomingCmd1:=FALSE;
			OP70_Homing_Seq:=75;
		END_IF

  75:	IF OP70_GIUDE_GRP_ctrl.Axis_In_Home AND OP70_GIUDE_GRP_ctrl.Axis_Home_Done THEN
	  		OP70_GIUDE_GRP_ctrl.Bsethome:=0;
			OP70_Homing_Seq:=80;
		ELSE
			OP70_GIUDE_GRP_ctrl.Bsethome:=1;
  		END_IF
		
   80:	OP70_Homing_Seq:=0;
   		CR70_LH_Rej_Cyl.HomingCmd1:=FALSE;
   		CR70_RH_Rej_Cyl.HomingCmd1:=FALSE;
		OP70_HomeRunning:=FALSE;
		OP70_HMI_Homing:=FALSE;
END_CASE


Homing_Check_Timer(IN:=(OP70_Homing_Seq=40),PT:=T#2S);

IF Homing_Check_Timer.Q THEN
	OP70_Gripper_LH_Gripper_ctrl.Reference_Start:=Pulse_Block.Q1Hz ;
	OP70_Gripper_RH_Gripper_ctrl.Reference_Start:=Pulse_Block.Q1Hz ;
END_IF

END_PROGRAM

// ---- POUs/Programs/OP70/OP70_Conveyor_Cam_Seq.TcPOU
PROGRAM OP70_Conveyor_Cam_Seq
VAR
	OP70_Conveyor	: Servo_Conveyor_FB;
	Conv_Cam_Step: INT;
	OP70_Camera_Trigger: BOOL;
	OP70_Miss_Trigger: BOOL;
	OP70_LH_Camera_OK: BOOL;
	OP70_LH_Camera_NOK: BOOL;
	OP70_RH_Camera_OK: BOOL;
	OP70_RH_Camera_NOK: BOOL;
	OP70_LH_Clr_OK: BOOL;
	OP70_RH_Clr_OK: BOOL;
	OP70_LH_Size_NOK: BOOL;
	OP70_RH_Size_NOK: BOOL;
	OP70_Size_Rej: BOOL;
	OP70_LH_Clr_NOK : BOOL;
	OP70_RH_Clr_NOK	: BOOL;
	OP70_Size_Rej_Complete: BOOL;
	Conveyor_Track_Delay: TON;
	Conveyor_Track_OFF_Delay: TON;
	Conveyor_Velocity_mode : BOOL;
	Servo_Conti_Run			: BOOL;
	Temp_Counter_LH			: UDINT;
	Temp_Counter_RH			: UDINT;
	//OP70_Camera_Trigger: BOOL;
	OP70_LH_Size_OK: BOOL;
	OP70_RH_Size_OK: BOOL;
	OP70_Camera_Trigger_Ack : BOOL;
	Toggle_Pos_LH : R_TRIG;
	Toggle_Neg_LH : F_TRIG;
	Toggle_Pos_RH : R_TRIG;
	Toggle_Neg_RH : F_TRIG;
	LH_Cam_Completed : BOOL;
	RH_Cam_Completed : BOOL;
	Drum_Jam_Timer	 : TON;
	Conv_Step_no: INT;
	OP70_Camera_Bypass : BOOL;
	Control : BOOL;
END_VAR


Toggle_Pos_LH(CLK:=OP70_Camera_FB.OP70_LH_Inspection_Status.Inspection_Completed);
Toggle_Neg_LH(CLK:=OP70_Camera_FB.OP70_LH_Inspection_Status.Inspection_Completed);
Toggle_Pos_RH(CLK:=OP70_Camera_FB.OP70_RH_Inspection_Status.Inspection_Completed);
Toggle_Neg_RH(CLK:=OP70_Camera_FB.OP70_RH_Inspection_Status.Inspection_Completed);

IF Toggle_Pos_LH.Q OR Toggle_Neg_LH.Q THEN
	LH_Cam_Completed:=1;	
END_IF
IF Toggle_Pos_RH.Q OR Toggle_Neg_RH.Q THEN
	RH_Cam_Completed:=1;	
END_IF


IF MANUAL_SELECTED AND OP70_ManualSelected THEN               
	IF I70_DRUM_CONV_REV_I308_3 THEN
		SR70_Conv_servo_status.targetVelocity:=OP70_Conv_Rev_Speed_6_3;
		SR70_Conv_servo_status.moveVelocity:=I70_DRUM_CONV_REV_I308_3;
 	ELSIF I70_DRUM_CONV_FWD_I308_4 THEN
		SR70_Conv_servo_status.targetVelocity:=OP70_Conv_Fwd_Speed_7_89;
		SR70_Conv_servo_status.moveVelocity:=I70_DRUM_CONV_FWD_I308_4;	
	ELSE 	
		SR70_Conv_servo_status.moveVelocity:=0;   	
	END_IF  	
END_IF

OP70_Model:=Model;

IF OP70_Model='6.3' THEN
	OP70_Conv_Fwd_Time:=OP70_Conv_Fwd_Time_6_3;
	OP70_Conv_Rev_Time:=OP70_Conv_Rev_Time_6_3;
	OP70_Conveyor_FWD_Speed:= OP70_Conv_Fwd_Speed_6_3;
	OP70_Conveyor_REV_Speed:= OP70_Conv_Rev_Speed_6_3;
END_IF

IF OP70_Model='7.89' THEN
	OP70_Conv_Fwd_Time:=OP70_Conv_Fwd_Time_7_89;
	OP70_Conv_Rev_Time:=OP70_Conv_Rev_Time_7_89;
	OP70_Conveyor_FWD_Speed:= OP70_Conv_Fwd_Speed_7_89;
	OP70_Conveyor_REV_Speed:= OP70_Conv_Rev_Speed_7_89;
END_IF

Conveyor_Velocity_mode:=1;

OP70_Conveyor(
	Conveyor_Prgrm_Start:= OP70_Conveyor_ON AND OP70_AutoRunning, 
	Conveyor_Prgrm_Reset:= , 
	Conveyor_Continuous_Run:= Servo_Conti_Run, 
	Conveyor_FWD_Position	:= OP70_Conv_Fwd_Pos,
    Conveyor_REV_Position	:= OP70_Conv_Rev_Pos,
    Velocity_mode			:= Conveyor_Velocity_mode,	
	Track_Overflow := Conveyor_Track_OFF_Delay.Q, 
    Track_Sensor_FB := Conveyor_Track_Delay.Q,	
	Camera_Trigger_OK := OP70_Camera_Done OR OP70_Camera_Bypass, 
	Fwd_Time_IP:= OP70_Conv_Fwd_Time, 
	Rev_Time_IP:= OP70_Conv_Rev_Time, 
	Conveyor_FWD_Speed:=OP70_Conveyor_FWD_Speed , 
	Conveyor_REV_Speed:=OP70_Conveyor_REV_Speed , 
	LH_Work_Sensor:=CR70_LH_Rej_Cyl.Sensor2 , 
	LH_Home_Sensor:=CR70_LH_Rej_Cyl.Sensor1 , 
	RH_Work_Sensor:=CR70_RH_Rej_Cyl.Sensor2 , 
	RH_Home_Sensor:=CR70_RH_Rej_Cyl.Sensor1 , 
	LH_Camera_OK:=  OP70_RH_Camera_OK OR OP70_Camera_Bypass, 
	LH_Camera_NOK:= OP70_RH_Camera_NOK, 
	RH_Camera_OK:=  OP70_LH_Camera_OK OR OP70_Camera_Bypass, 
	RH_Camera_NOK:= OP70_LH_Camera_NOK, 
	Camera_trigger:= OP70_Camera_Trigger,
	Camera_Trigger_Ack=> OP70_Camera_Trigger_Ack,
	Step_Num => Conv_Step_no,
	Drum_ON=> O70_DRUM_MTR_FWD_Q307_1, 
	LH_Work_Coil=>CR70_LH_Rej_Cyl.AutoCmd2 , 
	LH_Home_Coil=>CR70_LH_Rej_Cyl.AutoCmd1 , 
	RH_Work_Coil=>CR70_RH_Rej_Cyl.AutoCmd2,
	RH_Home_Coil=>CR70_RH_Rej_Cyl.AutoCmd1,
	Ready_to_Pick=> OP70_pick_ready , 
	One_Cycle		:= OP70_One_Cycle,	
	Pick_Done:=     OP70_pick_done , 
	Conveyor_Servo_Control_Structure:= SR70_CONV_servo_ctrl );

Conveyor_Track_Delay(IN:= NOT I70_DRUM_FEED_CONV1_OVERFLW_I1110_2 OR NOT I70_DRUM_FEED_CONV2_OVERFLW_I1110_3,PT:=INT_TO_TIME(OP70_Drum_ON_Time));	
Conveyor_Track_OFF_Delay(IN:=I70_DRUM_FEED_CONV1_OVERFLW_I1110_2 AND I70_DRUM_FEED_CONV2_OVERFLW_I1110_3,PT:=INT_TO_TIME(OP70_Drum_OFF_Time)); //  
	
IF 	OP70_AutoRunning THEN
	IF Conveyor_Track_OFF_Delay.Q THEN
		O70_DRUM_MTR_FWD_Q307_1:=0;
	END_IF
	//IF Conveyor_Track_Delay.Q THEN
	//	O70_DRUM_MTR_FWD_Q307_1:=1;
	//END_IF
	O70_AIR_PURGE_ON_Q1153_6:=1;
	O70_DRUM_RUN_IND_Q307_5 :=O70_DRUM_MTR_FWD_Q307_1;
ELSE
	O70_DRUM_MTR_FWD_Q307_1:=I70_DRUM_OFF_ON_I308_2;
	O70_DRUM_RUN_IND_Q307_5:=I70_DRUM_OFF_ON_I308_2;
	O70_AIR_PURGE_ON_Q1153_6:=I70_DRUM_OFF_ON_I308_2;
END_IF	

IF (NOT OP70_AutoRunning OR (NOT OP70_LH_Camera_Online OR NOT OP70_RH_Camera_Online)) AND NOT OP70_Camera_Bypass THEN
	Conv_Cam_Step:=10;
END_IF 

CASE Conv_Cam_Step OF
	10: 	OP70_LH_Camera_OK :=0;
            OP70_LH_Camera_NOK:=0;
	        OP70_RH_Camera_OK :=0;
	        OP70_RH_Camera_NOK:=0;	
			LH_Cam_Completed  :=0;
			RH_Cam_Completed  :=0;		
			OP70_Camera_Done	:=0;
			OP70_LH_Clr_OK 		:=0;
		    OP70_RH_Clr_OK 		:=0;		
			OP70_LH_Size_OK		:=0;
		    OP70_RH_Size_OK		:=0;	
			Conv_Cam_Step		:=11;	
	
	11: IF ((OP70_Camera_Trigger AND (NOT OP70_Camera_Done)) OR OP70_Miss_Trigger) AND NOT OP70_Camera_Bypass THEN
			OP70_LH_Camera_Trigger:=1;
			OP70_RH_Camera_Trigger:=1;
			Conv_Cam_Step		  :=15;	
		END_IF

	15:	IF LH_Cam_Completed AND RH_Cam_Completed THEN// (NOT OP70_LH_Camera_Trigger) AND (NOT OP70_RH_Camera_Trigger) THEN //(Temp_Counter_LH<OP70_Camera_FB.OP70_LH_Acquisition_ID AND Temp_Counter_RH<OP70_Camera_FB.OP70_RH_Acquisition_ID )THEN
			OP70_LH_Camera_Trigger:=0;
			OP70_RH_Camera_Trigger:=0;
			OP70_Camera_Trigger :=0;
			OP70_Miss_Trigger	:=0;
			Conv_Cam_Step:=25;
		END_IF  
	   
	25: IF OP70_Camera_FB.OP70_LH_Cam_Result[0]=1 AND OP70_Camera_FB.OP70_RH_Cam_Result[0]=1 THEN
			OP70_LH_Camera_OK:=1;
			OP70_RH_Camera_OK:=1;
			Conv_Cam_Step    :=50;
		ELSIF (OP70_Camera_FB.OP70_LH_Cam_Result[2]<>1 OR OP70_Camera_FB.OP70_RH_Cam_Result[2]<>1) THEN	
			OP70_One_Cycle  :=1;
			Conv_Cam_Step   :=50;
		ELSIF (OP70_Camera_FB.OP70_LH_Cam_Result[1]=1 OR OP70_Camera_FB.OP70_RH_Cam_Result[1]=1) AND (OP70_Camera_FB.OP70_LH_Cam_Result[2]=1 AND OP70_Camera_FB.OP70_RH_Cam_Result[2]=1) THEN			
			IF OP70_Camera_FB.OP70_LH_Cam_Result[0]=1 THEN
				OP70_LH_Camera_OK:=1;
			END_IF
			IF OP70_Camera_FB.OP70_RH_Cam_Result[0]=1 THEN
				OP70_RH_Camera_OK:=1;
			END_IF
			Conv_Cam_Step:=30;
		END_IF	
			
   30: 	IF OP70_Camera_FB.OP70_LH_Cam_Result[1]=1 THEN
	   		OP70_LH_Camera_NOK:=1;
  	    END_IF
		IF OP70_Camera_FB.OP70_RH_Cam_Result[1]=1 THEN
	   		OP70_RH_Camera_NOK:=1;
  	    END_IF
		Conv_Cam_Step:=50;
		
   50:  OP70_Camera_Done:=1;
   		Temp_Counter_LH:=OP70_Camera_FB.OP70_LH_Acquisition_ID;
		Temp_Counter_RH:=OP70_Camera_FB.OP70_RH_Acquisition_ID;
		IF Conv_Step_no>75 THEN
			Conv_Cam_Step   :=10;
			OP70_Camera_Done:=0;
		END_IF
   	    
END_CASE

IF OP70_AutoRunning AND Control THEN
	Drum_Jam_Timer(IN:=(NOT I70_DRUM_FEED_CONV1_OVERFLW_I1110_2)OR(NOT I70_DRUM_FEED_CONV1_OVERFLW_I1110_2)); 
	Drum_Jam_Timer(PT:=T#40S);
	IF Drum_Jam_Timer.Q THEN
		OP70_ErrorActive:=1;
	END_IF
END_IF



(*	30: IF OP70_Camera_FB.OP70_LH_Cam_Result[4]<>1 OR OP70_Camera_FB.OP70_RH_Cam_Result[4]<>1 THEN
		 	IF OP70_Camera_FB.OP70_LH_Cam_Result[4]<>1 THEN
				OP70_LH_Size_NOK:=1;
			END_IF
		 	IF OP70_Camera_FB.OP70_RH_Cam_Result[4]<>1 THEN
				OP70_RH_Size_NOK:=1;
			END_IF
		    OP70_Size_Rej:=1;
		    IF OP70_Size_Rej_Complete THEN
			    OP70_One_Cycle:=1;
			    Conv_Cam_Step:=10;
		    END_IF	 
		ELSIF OP70_Camera_FB.OP70_LH_Cam_Result[4]=1 AND OP70_Camera_FB.OP70_RH_Cam_Result[4]=1 THEN
			 OP30_LH_Size_OK:= 1;
		     OP30_RH_Size_OK:= 1;
			 Conv_Cam_Step:=40;
		END_IF
		
	40: IF OP70_Camera_FB.OP70_LH_Cam_Result[3]<>1 OR OP70_Camera_FB.OP70_RH_Cam_Result[3]<>1 THEN
		 	IF OP70_Camera_FB.OP70_LH_Cam_Result[3]<>1 THEN
				OP70_LH_Clr_NOK:=1;
				OP70_LH_Camera_NOK:=1;
			END_IF
		 	IF OP70_Camera_FB.OP70_RH_Cam_Result[3]<>1 THEN
				OP70_RH_Clr_NOK:=1;
				OP70_RH_Camera_NOK:=1;
			END_IF
			Conv_Cam_Step  :=70;
		ELSIF OP70_Camera_FB.OP70_LH_Cam_Result[3]=1 AND OP70_Camera_FB.OP70_RH_Cam_Result[3]=1 THEN
			 OP70_LH_Clr_OK :=1;
		     OP70_RH_Clr_OK :=1;
			 Conv_Cam_Step  :=50;
		END_IF 
*)

END_PROGRAM

// ---- POUs/Programs/OP70/OP70_CONVEYOR.TcPOU
PROGRAM OP70_CONVEYOR
VAR
	con_step_no : INT;
	cam_trig : BOOL;
	cam_ok : BOOL;
	LH_Cam_OK : BOOL;
	RH_Cam_OK : BOOL;
	t1: ton;
	t2: ton;
	t3: ton;
	t4: ton;
	
	temp: BOOL;
	check:BOOL;
	check1:ton;
	fwd_time : INT :=500;
	rev_time : INT :=500;	
	count_nok :INT;
	forward: BOOL;
	reverse: BOOL;

	temp1: BOOL;
	temp2: BOOL;
	
	LH_Cyl_Delay : TON;
	RH_Cyl_Delay : TON;
	temp_3: BOOL;
END_VAR

IF (NOT OP70_AutoSelected OR OP70_ErrorActive ) THEN
	//SR70_CONV_servo_ctrl.VELmove_Start:=FALSE;
	forward:=FALSE;
	reverse:=FALSE;
	con_step_no:= 10;
END_IF	



IF MANUAL_SELECTED AND OP70_ManualSelected THEN               
	IF I70_DRUM_CONV_REV_I308_3 THEN
		SR70_Conv_servo_status.targetVelocity:=OP70_Conv_Rev_Speed_6_3;
		SR70_CONV_servo_ctrl.VELmove_Start:=I70_DRUM_CONV_REV_I308_3;
 	ELSIF I70_DRUM_CONV_FWD_I308_4 THEN
		SR70_Conv_servo_status.targetVelocity:=OP70_Conv_Fwd_Speed_7_89;
		SR70_CONV_servo_ctrl.VELmove_Start:=I70_DRUM_CONV_FWD_I308_4;	
	ELSE 	
		SR70_CONV_servo_ctrl.VELmove_Start:=0;   	
	END_IF  	
END_IF
                


CASE con_step_no OF
		10: IF (OP70_AutoSelected) THEN		// Check Automode Selected
				con_step_no:=65;
	        END_IF
		   
        65:	forward:=TRUE;
			SR70_CONV_servo_ctrl.Velocity:= OP70_Conveyor_Speed;
			SR70_CONV_servo_ctrl.VELmove_Start:=TRUE;	
			IF t2.Q THEN
    			forward:=FALSE;
				SR70_CONV_servo_ctrl.VELmove_Start:=FALSE;
				con_step_no:= 70;
			END_IF
		  
		70: IF NOT SR70_CONV_servo_ctrl.VELmove_Start THEN
			  cam_trig :=TRUE;
			  IF t1.Q THEN
				con_step_no:= 75;
			  END_IF
			END_IF	
					
		75:	IF cam_ok AND NOT SR70_CONV_servo_ctrl.VELmove_Start AND SR70_CONV_servo_ctrl.Axis_ready THEN
				IF LH_Cam_OK AND RH_Cam_OK THEN
				 con_step_no:= 90;
				 fwd_time:=OP70_Conv_Fwd_Time_6_3;
				 count_nok:=0;	
				ELSIF (NOT LH_Cam_OK OR NOT RH_Cam_OK) AND count_nok<5 THEN
				 count_nok := count_nok +1;
				 con_step_no:= 76;	
				ELSIF count_nok>=5 THEN
	             fwd_time:=7000;
				 con_step_no:= 80; 
				END_IF
			END_IF	
			
		76:	 IF NOT LH_Cam_OK AND NOT SR70_CONV_servo_ctrl.VELmove_Start THEN
				CR70_LH_Rej_Cyl.AutoCmd1:=0;
				CR70_LH_Rej_Cyl.AutoCmd2:=TRUE;
				con_step_no:= 78;
			ELSIF LH_Cam_OK THEN
				con_step_no:= 77;
			END_IF	
			
	   78:	IF I70_LH_REJ_CYL_REV_I1110_5 AND LH_Cyl_Delay.Q THEN
				CR70_LH_Rej_Cyl.AutoCmd1:=1;
				CR70_LH_Rej_Cyl.AutoCmd2:=0;
				con_step_no:= 79;					
			END_IF
			
	   79: IF I70_LH_REJ_CYL_FWD_I1110_4 AND count_nok<5 AND NOT CR70_LH_Rej_Cyl.AutoCmd2 THEN
				CR70_LH_Rej_Cyl.AutoCmd1:=0;
				con_step_no:= 77;
		   END_IF
           IF count_nok>5 THEN
			 fwd_time:=7000;
		     con_step_no:= 77;	
		   END_IF

			
	   77:	IF NOT RH_Cam_OK AND NOT SR70_CONV_servo_ctrl.VELmove_Start THEN	
				CR70_RH_Rej_Cyl.AutoCmd1:=0;
				CR70_RH_Rej_Cyl.AutoCmd2:=TRUE;				
				con_step_no:= 81;
			ELSIF RH_Cam_OK THEN
				con_step_no:= 80;
			END_IF

		81:	    IF  I70_RH_REJ_CYL_REV_I1110_7 AND RH_Cyl_Delay.Q THEN
					CR70_RH_Rej_Cyl.AutoCmd1:=1;
					CR70_RH_Rej_Cyl.AutoCmd2:=0;	
					con_step_no:= 82;			
				END_IF		
				
		82: 	IF I70_RH_REJ_CYL_FWD_I1110_6 AND count_nok<5 AND NOT CR70_RH_Rej_Cyl.AutoCmd2 THEN
					CR70_RH_Rej_Cyl.AutoCmd1:=0;					
					//fwd_time:=OP70_Conv_Fwd_Time_6_3;			  
				END_IF
				IF count_nok>5 THEN
					fwd_time:=7000;
				    con_step_no:= 80;	
				END_IF
	
		80: 	IF fwd_time=7000 THEN
			       count_nok:=0;	
				END_IF
                SR70_CONV_servo_ctrl.Velocity:= OP70_Conveyor_Speed;				
				forward:=TRUE;
				SR70_CONV_servo_ctrl.VELmove_Start:=TRUE;
				IF t2.Q THEN
    				forward:=FALSE;
					con_step_no:= 70;
					SR70_CONV_servo_ctrl.VELmove_Start:=FALSE;				
				END_IF
		        
		90: 	SR70_CONV_servo_ctrl.Velocity:= OP70_Conveyor_Speed;
				reverse:=TRUE;
				SR70_CONV_servo_ctrl.VELmove_Start:=TRUE;	
				IF t3.Q THEN				
 					reverse:=FALSE;
					SR70_CONV_servo_ctrl.VELmove_Start:=FALSE;
					con_step_no:= 100;				
				END_IF		
				
		100: OP70_pick_ready:=TRUE;
			 IF OP70_pick_done OR temp_3 THEN
				 OP70_pick_ready :=FALSE;
				 OP70_pick_done:=FALSE;
				 con_step_no:= 80;
			 END_IF
			 		
				
END_CASE

t1(IN:=cam_trig ,PT:=T#700MS);
IF cam_trig AND con_step_no=70  THEN // Reset for next cycle
	cam_ok:=FALSE;
	LH_Cam_OK:=0;
	RH_Cam_OK:=0;
END_IF

IF t1.Q THEN //Result updating from Camera
	cam_ok:=TRUE;
	LH_Cam_OK:=temp1;
	RH_Cam_OK:=temp2;
	cam_trig :=FALSE;
END_IF


t2(IN:=forward ,PT:=INT_TO_TIME(fwd_time));
t3(IN:=reverse ,PT:=INT_TO_TIME(rev_time));
t4(IN:=cam_ok,PT:=T#1S);

LH_Cyl_Delay(IN:= I70_LH_REJ_CYL_FWD_I1110_4 ,PT:=T#300MS);
RH_Cyl_Delay(IN:= I70_RH_REJ_CYL_FWD_I1110_6 ,PT:=T#300MS);

END_PROGRAM

// ---- POUs/Programs/OP80/OP80_MAIN.TcPOU
PROGRAM OP80_MAIN
VAR
	OP80_Modeselection_FB: Mode_Selection_Block1;	
//	OP80_Cycle_Time: Cycle_Time_FB;
	reset: BOOL;
	Gen_Timer: TON;
END_VAR

// Function Calling

OP80_Manual();
OP80_AUTOSEQUENCE();
OP80_Error();
OP80_Initialization_Seq();
op80_toolchangeover ();
//MOdeselection From HMI

